Yaskawa INFORM job: CPRINT3D2.JBI

/JOB
//NAME CPRINT3D2
//POS
///NPOS 999,0,0,0,0,0
///TOOL 9
///POSTYPE PULSE
///PULSE
C00000=28439,52447,-122346,62432,-118756,-94394,0
C00001=28774,52172,-123325,61938,-118477,-94718,0
C00002=28786,52165,-123350,61921,-118471,-94727,0
C00003=28820,52146,-123417,61875,-118455,-94751,0
C00004=28874,52134,-123462,61810,-118455,-94770,0
C00005=28928,52121,-123507,61744,-118455,-94790,0
C00006=29088,52031,-123833,61527,-118375,-94904,0
C00007=29175,51999,-123949,61415,-118355,-94948,0
C00008=29421,52045,-123790,61164,-118501,-94935,0
C00009=29495,52038,-123817,61080,-118514,-94952,0
C00010=29569,52031,-123842,60995,-118527,-94969,0
C00011=29587,52039,-123815,60978,-118545,-94964,0
C00012=29506,52029,-123847,61064,-118504,-94962,0
C00013=29829,52073,-123695,60727,-118672,-94961,0
C00014=29932,52093,-123628,60621,-118733,-94956,0
C00015=29996,52105,-123587,60557,-118771,-94953,0
C00016=30178,52149,-123434,60375,-118894,-94933,0
C00017=30236,52166,-123374,60319,-118938,-94924,0
C00018=30330,52195,-123273,60228,-119011,-94908,0
C00019=30378,52209,-123223,60182,-119047,-94901,0
C00020=30588,52286,-122956,59985,-119227,-94854,0
C00021=30620,52321,-122833,59966,-119289,-94824,0
C00022=30635,52338,-122772,59957,-119320,-94809,0
C00023=49239,53005,-120913,62324,-119586,-94086,0
C00024=49295,53006,-120913,62261,-119605,-94093,0
C00025=49352,53006,-120913,62199,-119626,-94101,0
C00026=49357,53007,-120910,62194,-119628,-94101,0
C00027=49400,53018,-120873,62152,-119658,-94096,0
C00028=49596,53097,-120607,61973,-119832,-94048,0
C00029=49625,53101,-120595,61943,-119847,-94048,0
C00030=49712,53113,-120558,61852,-119893,-94050,0
C00031=49739,53123,-120523,61827,-119916,-94044,0
C00032=49769,53136,-120482,61800,-119943,-94037,0
C00033=50226,53391,-119629,61417,-120443,-93863,0
C00034=50247,53407,-119575,61401,-120472,-93851,0
C00035=50264,53421,-119528,61390,-120497,-93840,0
C00036=50275,53464,-119383,61398,-120558,-93801,0
C00037=50279,53479,-119335,61401,-120579,-93788,0
C00038=50414,53586,-118980,61302,-120768,-93708,0
C00039=50453,53638,-118808,61285,-120851,-93666,0
C00040=50279,53728,-118502,61520,-120908,-93555,0
C00041=50270,53764,-118384,61547,-120951,-93521,0
C00042=50261,53800,-118264,61574,-120995,-93487,0
C00043=50239,53805,-118247,61601,-120993,-93478,0
C00044=50284,53772,-118356,61536,-120967,-93516,0
C00045=50093,53900,-117929,61808,-121064,-93368,0
C00046=50021,53939,-117796,61906,-121089,-93320,0
C00047=49977,53963,-117716,61966,-121103,-93291,0
C00048=49831,54030,-117493,62159,-121135,-93207,0
C00049=49779,54050,-117426,62226,-121141,-93181,0
C00050=49693,54082,-117318,62336,-121150,-93137,0
C00051=49650,54098,-117264,62391,-121153,-93116,0
C00052=49433,54167,-117032,62662,-121159,-93019,0
C00053=49353,54169,-117024,62751,-121131,-93005,0
C00054=49313,54170,-117021,62795,-121118,-92998,0
C00055=49104,54236,-116799,63057,-121120,-92904,0
C00056=49064,54233,-116808,63099,-121101,-92901,0
C00057=40018,60732,-97213,75689,-122654,-85947,0
C00058=40054,60785,-97067,75678,-122711,-85911,0
C00059=40032,60817,-96978,75714,-122721,-85882,0
C00060=40014,60842,-96907,75743,-122726,-85859,0
C00061=39996,60867,-96836,75772,-122733,-85836,0
C00062=39979,60893,-96765,75801,-122740,-85813,0
C00063=39961,60918,-96694,75831,-122747,-85790,0
C00064=39951,60933,-96653,75848,-122750,-85776,0
C00065=39894,60999,-96467,75934,-122761,-85715,0
C00066=39865,61033,-96374,75978,-122767,-85684,0
C00067=39823,61077,-96250,76039,-122770,-85642,0
C00068=39761,61137,-96083,76128,-122772,-85585,0
C00069=39725,61172,-95986,76179,-122773,-85552,0
C00070=39700,61192,-95929,76214,-122772,-85532,0
C00071=39675,61212,-95873,76248,-122770,-85512,0
C00072=39649,61232,-95816,76282,-122768,-85492,0
C00073=39624,61253,-95760,76316,-122765,-85472,0
C00074=39598,61273,-95703,76351,-122764,-85452,0
C00075=39580,61287,-95663,76375,-122762,-85438,0
C00076=39514,61268,-95714,76432,-122709,-85443,0
C00077=23111,61906,-93699,72648,-125561,-85469,0
C00078=23063,61952,-93573,72718,-125566,-85425,0
C00079=23022,61942,-93597,72755,-125534,-85425,0
C00080=22989,61935,-93618,72784,-125507,-85426,0
C00081=22956,61927,-93639,72813,-125482,-85426,0
C00082=22923,61919,-93660,72842,-125456,-85426,0
C00083=22890,61912,-93680,72871,-125430,-85426,0
C00084=22871,61907,-93692,72888,-125415,-85427,0
C00085=22781,61878,-93772,72962,-125340,-85434,0
C00086=22736,61863,-93811,73000,-125302,-85438,0
C00087=22678,61841,-93871,73047,-125250,-85445,0
C00088=22634,61823,-93921,73081,-125210,-85452,0
C00089=22547,61786,-94022,73149,-125129,-85466,0
C00090=22530,61777,-94046,73161,-125113,-85470,0
C00091=22501,61761,-94089,73183,-125083,-85477,0
C00092=22472,61745,-94132,73204,-125055,-85484,0
C00093=22442,61729,-94175,73225,-125025,-85492,0
C00094=22413,61713,-94218,73247,-124996,-85499,0
C00095=22377,61694,-94271,73273,-124959,-85508,0
C00096=22378,61632,-94442,73241,-124916,-85557,0
C00097=22087,61535,-94704,73483,-124670,-85584,0
C00098=22099,61276,-95420,73344,-124490,-85788,0
C00099=22144,61093,-95926,73210,-124385,-85939,0
C00100=22157,61056,-96029,73179,-124365,-85970,0
C00101=22183,60982,-96235,73117,-124326,-86033,0
C00102=22199,60937,-96360,73079,-124302,-86071,0
C00103=22261,60808,-96718,72954,-124244,-86182,0
C00104=22286,60767,-96832,72909,-124228,-86219,0
C00105=22328,60702,-97015,72836,-124204,-86278,0
C00106=22437,60560,-97411,72657,-124163,-86407,0
C00107=22476,60515,-97537,72596,-124151,-86449,0
C00108=22493,60521,-97521,72582,-124165,-86447,0
C00109=22439,60543,-97459,72646,-124151,-86421,0
C00110=22493,60521,-97521,72582,-124165,-86447,0
C00111=22546,60499,-97583,72517,-124180,-86474,0
C00112=22546,60446,-97605,72528,-124197,-86456,0
C00113=40139,58675,-102915,74674,-121313,-87587,0
C00114=46748,54147,-116851,65625,-120206,-92552,0
C00115=46543,53843,-117842,65707,-119772,-92808,0
C00116=46527,53787,-118025,65698,-119701,-92859,0
C00117=46489,53721,-118242,65709,-119608,-92917,0
C00118=46439,53445,-119159,65637,-119259,-93176,0
C00119=46497,53175,-120068,65451,-118951,-93447,0
C00120=46664,52922,-120936,65152,-118694,-93722,0
C00121=46813,52797,-121368,64933,-118587,-93867,0
C00122=31513,53470,-118728,59563,-121334,-93793,0
C00123=31001,53645,-118138,60213,-121386,-93553,0
C00124=30898,53667,-118063,60337,-121380,-93517,0
C00125=30785,53702,-117945,60479,-121384,-93467,0
C00126=30275,53799,-117618,61087,-121323,-93299,0
C00127=29739,53845,-117457,61698,-121183,-93173,0
C00128=29195,53838,-117469,62291,-120970,-93095,0
C00129=28904,53806,-117570,62595,-120820,-93080,0
C00130=24595,59466,-100389,69956,-124580,-87578,0
C00131=25008,59807,-99429,69702,-125092,-87378,0
C00132=25274,60150,-98469,69602,-125526,-87155,0
C00133=25393,60407,-97751,69612,-125804,-86976,0
C00134=25484,60702,-96928,69671,-126098,-86762,0
C00135=29736,55171,-113211,83941,-113532,-89553,0
C00136=29662,55374,-112578,84077,-113612,-89348,0
C00137=37622,58900,-102216,77312,-120074,-87045,0
C00138=38136,58667,-102898,76698,-120202,-87311,0
C00139=38618,58542,-103267,76159,-120381,-87482,0
C00140=38958,58510,-103367,75801,-120545,-87556,0
C00141=39335,58507,-103383,75417,-120750,-87612,0
C00142=39839,58581,-103180,74938,-121078,-87622,0
C00143=40057,58649,-102988,74746,-121249,-87596,0
C00144=40323,59480,-100616,74849,-122006,-86947,0
C00145=47960,54217,-116657,64337,-120759,-92670,0
C00146=47759,54094,-117052,64499,-120535,-92753,0
C00147=47571,53923,-117607,64624,-120258,-92884,0
C00148=47451,53740,-118207,64669,-119993,-93039,0
C00149=47440,53697,-118347,64661,-119936,-93078,0
C00150=47411,53644,-118524,64668,-119860,-93124,0
C00151=47383,53460,-119134,64613,-119625,-93296,0
C00152=47428,53280,-119739,64481,-119418,-93476,0
C00153=47544,53111,-120315,64275,-119246,-93657,0
C00154=47729,52958,-120841,64001,-119115,-93834,0
C00155=48077,52776,-121476,63535,-118995,-94063,0
C00156=31284,52867,-120754,59528,-120418,-94315,0
C00157=31125,52990,-120334,59762,-120536,-94176,0
C00158=30851,53126,-119866,60129,-120633,-94006,0
C00159=30540,53231,-119506,60524,-120667,-93860,0
C00160=30461,53248,-119449,60619,-120661,-93833,0
C00161=30368,53276,-119352,60735,-120667,-93793,0
C00162=30024,53340,-119134,61143,-120629,-93682,0
C00163=29662,53370,-119026,61556,-120540,-93598,0
C00164=29294,53365,-119034,61959,-120400,-93547,0
C00165=28932,53327,-119157,62337,-120219,-93530,0
C00166=28454,53226,-119485,62815,-119916,-93555,0
C00167=23569,59757,-99551,71154,-124247,-87172,0
C00168=23875,59858,-99271,70890,-124500,-87143,0
C00169=24154,60011,-98844,70680,-124781,-87070,0
C00170=24390,60208,-98293,70538,-125074,-86955,0
C00171=24575,60444,-97635,70469,-125368,-86801,0
C00172=24652,60608,-97180,70473,-125544,-86687,0
C00173=24715,60805,-96632,70510,-125737,-86544,0
C00174=24738,61093,-95833,70634,-125978,-86325,0
C00175=24696,61382,-95035,70826,-126178,-86094,0
C00176=24554,61763,-93987,71167,-126386,-85776,0
C00177=37748,59756,-99783,77545,-120714,-86351,0
C00178=37941,59542,-100390,77263,-120685,-86553,0
C00179=38191,59363,-100905,76938,-120710,-86736,0
C00180=38484,59228,-101296,76587,-120785,-86889,0
C00181=38809,59142,-101548,76223,-120911,-87006,0
C00182=39022,59121,-101612,76000,-121015,-87054,0
C00183=39270,59119,-101622,75750,-121153,-87090,0
C00184=39611,59170,-101483,75429,-121382,-87097,0
C00185=39931,59273,-101196,75151,-121636,-87059,0
C00186=40250,59441,-100724,74904,-121937,-86968,0
C00187=48252,53381,-119424,63624,-119841,-93498,0
C00188=48319,53287,-119742,63507,-119744,-93599,0
C00189=48423,53202,-120032,63353,-119672,-93696,0
C00190=48560,53129,-120281,63169,-119626,-93786,0
C00191=48724,53072,-120481,62960,-119609,-93865,0
C00192=48911,53031,-120625,62736,-119619,-93932,0
C00193=48970,53025,-120648,62668,-119632,-93947,0
C00194=49055,53010,-120703,62567,-119640,-93974,0
C00195=49583,52969,-120858,61965,-119765,-94091,0
C00196=30650,52240,-122919,59933,-119302,-94827,0
C00197=30671,52456,-122162,60012,-119625,-94618,0
C00198=30635,52559,-121802,60100,-119762,-94512,0
C00199=30555,52657,-121463,60234,-119874,-94406,0
C00200=30442,52741,-121170,60399,-119956,-94309,0
C00201=30291,52816,-120911,60601,-120010,-94215,0
C00202=30117,52874,-120711,60820,-120030,-94134,0
C00203=30060,52885,-120668,60889,-120027,-94115,0
C00204=29985,52907,-120592,60981,-120032,-94083,0
C00205=29793,52942,-120471,61209,-120012,-94021,0
C00206=29591,52959,-120411,61441,-119965,-93976,0
C00207=29384,52956,-120415,61667,-119889,-93948,0
C00208=29182,52935,-120483,61879,-119790,-93939,0
C00209=28992,52896,-120614,62070,-119671,-93949,0
C00210=28820,52840,-120800,62233,-119536,-93978,0
C00211=28673,52771,-121036,62362,-119392,-94025,0
C00212=28639,52747,-121118,62389,-119347,-94043,0
C00213=28578,52715,-121227,62441,-119282,-94066,0
C00214=28300,52499,-121966,62647,-118894,-94240,0
C00215=22491,60387,-97770,72555,-124120,-86493,0
C00216=23005,60287,-98055,71986,-124342,-86658,0
C00217=23190,60283,-98068,71798,-124446,-86691,0
C00218=23373,60311,-97991,71625,-124573,-86699,0
C00219=23550,60370,-97828,71476,-124721,-86683,0
C00220=23711,60460,-97581,71356,-124883,-86640,0
C00221=23849,60576,-97258,71274,-125055,-86572,0
C00222=23959,60716,-96869,71234,-125228,-86481,0
C00223=23997,60795,-96649,71235,-125312,-86426,0
C00224=24033,60905,-96346,71254,-125418,-86347,0
C00225=24049,61076,-95874,71324,-125559,-86217,0
C00226=24026,61246,-95401,71434,-125676,-86080,0
C00227=23966,61411,-94947,71578,-125766,-85942,0
C00228=23918,61488,-94735,71665,-125796,-85875,0
C00229=23843,61582,-94474,71789,-125822,-85788,0
C00230=23703,61701,-94147,71990,-125826,-85672,0
C00231=23297,61933,-93506,72514,-125750,-85423,0
C00232=38223,60782,-96915,77518,-121658,-85582,0
C00233=38238,60338,-98154,77310,-121382,-85943,0
C00234=38280,60189,-98571,77204,-121311,-86070,0
C00235=38359,60050,-98964,77066,-121266,-86195,0
C00236=38471,59925,-99318,76900,-121249,-86312,0
C00237=38616,59820,-99617,76711,-121263,-86419,0
C00238=38786,59741,-99845,76506,-121308,-86508,0
C00239=38976,59689,-99994,76294,-121383,-86578,0
C00240=39078,59679,-100025,76188,-121435,-86601,0
C00241=39213,59678,-100031,76052,-121512,-86621,0
C00242=39412,59709,-99948,75866,-121648,-86625,0
C00243=39600,59770,-99778,75705,-121799,-86602,0
C00244=39770,59860,-99526,75576,-121960,-86554,0
C00245=39843,59919,-99363,75529,-122043,-86517,0
C00246=39927,60004,-99123,75483,-122152,-86460,0
C00247=40019,60149,-98717,75457,-122306,-86356,0
C00248=40157,60547,-97607,75500,-122662,-86056,0
C00249=49381,54129,-116981,62740,-121193,-92971,0
C00250=48940,54060,-117194,63191,-120943,-92965,0
C00251=48744,54006,-117364,63380,-120803,-92984,0
C00252=48573,53936,-117592,63534,-120652,-93024,0
C00253=48434,53851,-117867,63646,-120495,-93082,0
C00254=48330,53756,-118178,63714,-120340,-93155,0
C00255=48266,53654,-118511,63737,-120190,-93240,0
C00256=48259,53624,-118614,63730,-120149,-93269,0
C00257=48237,53581,-118753,63734,-120088,-93305,0
C00258=48225,53480,-119090,63701,-119957,-93400,0
C00259=48238,53430,-119257,63662,-119899,-93449,0
C00260=48103,53311,-119656,63755,-119698,-93544,0
C00261=49484,53946,-117583,62539,-121004,-93155,0
C00262=49610,53938,-117614,62397,-121039,-93182,0
C00263=49860,53921,-117674,62114,-121111,-93237,0
C00264=49874,53920,-117678,62098,-121114,-93240,0
C00265=49888,53919,-117682,62082,-121119,-93243,0
C00266=49902,53918,-117685,62067,-121122,-93246,0
C00267=49916,53917,-117690,62051,-121126,-93249,0
C00268=49930,53916,-117693,62035,-121129,-93252,0
C00269=49942,53915,-117698,62021,-121132,-93255,0
C00270=49954,53913,-117702,62006,-121135,-93259,0
C00271=49967,53912,-117707,61992,-121138,-93262,0
C00272=49979,53911,-117713,61978,-121141,-93265,0
C00273=49991,53909,-117717,61964,-121143,-93268,0
C00274=50002,53908,-117723,61951,-121145,-93271,0
C00275=50014,53906,-117729,61937,-121147,-93274,0
C00276=50026,53905,-117733,61924,-121150,-93278,0
C00277=50037,53903,-117739,61910,-121152,-93281,0
C00278=50049,53902,-117745,61896,-121154,-93284,0
C00279=50061,53900,-117749,61883,-121157,-93288,0
C00280=50123,53870,-117852,61799,-121141,-93325,0
C00281=50159,53851,-117915,61751,-121129,-93348,0
C00282=50186,53835,-117968,61714,-121119,-93367,0
C00283=50213,53819,-118021,61676,-121108,-93386,0
C00284=50240,53803,-118075,61639,-121097,-93405,0
C00285=50267,53787,-118127,61601,-121087,-93424,0
C00286=50285,53775,-118167,61575,-121078,-93437,0
C00287=50303,53763,-118207,61549,-121069,-93451,0
C00288=50319,53753,-118242,61528,-121060,-93464,0
C00289=50334,53742,-118278,61506,-121052,-93476,0
C00290=50349,53731,-118315,61484,-121044,-93488,0
C00291=50364,53721,-118350,61462,-121035,-93500,0
C00292=50379,53710,-118386,61441,-121027,-93512,0
C00293=50394,53699,-118422,61419,-121018,-93524,0
C00294=50407,53690,-118455,61400,-121010,-93536,0
C00295=50418,53681,-118485,61383,-121003,-93545,0
C00296=50429,53672,-118514,61366,-120995,-93555,0
C00297=50441,53663,-118543,61350,-120988,-93566,0
C00298=50450,53655,-118572,61335,-120980,-93575,0
C00299=50460,53646,-118601,61320,-120972,-93584,0
C00300=50470,53637,-118630,61305,-120964,-93594,0
C00301=50479,53629,-118658,61290,-120957,-93603,0
C00302=50489,53620,-118686,61276,-120949,-93613,0
C00303=50498,53613,-118714,61262,-120941,-93621,0
C00304=50506,53605,-118738,61250,-120935,-93629,0
C00305=50513,53598,-118762,61238,-120928,-93637,0
C00306=50521,53591,-118785,61227,-120921,-93645,0
C00307=50527,53584,-118808,61216,-120914,-93652,0
C00308=50534,53578,-118831,61205,-120907,-93659,0
C00309=50544,53567,-118864,61189,-120898,-93670,0
C00310=50538,53559,-118892,61192,-120885,-93677,0
C00311=50531,53550,-118923,61195,-120870,-93684,0
C00312=50524,53541,-118954,61199,-120856,-93692,0
C00313=50517,53531,-118985,61202,-120841,-93699,0
C00314=50509,53522,-119015,61206,-120826,-93707,0
C00315=50500,53511,-119050,61211,-120808,-93715,0
C00316=50491,53501,-119085,61216,-120791,-93724,0
C00317=50481,53491,-119119,61222,-120774,-93732,0
C00318=50472,53480,-119154,61227,-120757,-93740,0
C00319=50463,53470,-119188,61233,-120739,-93748,0
C00320=50453,53459,-119223,61238,-120722,-93757,0
C00321=50444,53449,-119257,61243,-120706,-93765,0
C00322=50433,53438,-119293,61250,-120688,-93773,0
C00323=50422,53428,-119328,61257,-120669,-93782,0
C00324=50411,53417,-119364,61264,-120651,-93790,0
C00325=50396,53404,-119408,61274,-120629,-93800,0
C00326=50378,53388,-119460,61286,-120602,-93812,0
C00327=50360,53372,-119512,61299,-120574,-93823,0
C00328=50342,53357,-119564,61312,-120548,-93836,0
C00329=50323,53341,-119616,61324,-120520,-93847,0
C00330=50301,53324,-119674,61341,-120489,-93860,0
C00331=50271,53302,-119744,61364,-120450,-93876,0
C00332=50234,53278,-119827,61392,-120404,-93894,0
C00333=50198,53253,-119910,61421,-120358,-93912,0
C00334=50189,53251,-119917,61430,-120352,-93912,0
C00335=50178,53249,-119924,61441,-120345,-93912,0
C00336=50167,53246,-119932,61452,-120338,-93913,0
C00337=50156,53244,-119939,61464,-120332,-93913,0
C00338=50144,53242,-119947,61475,-120325,-93914,0
C00339=50133,53239,-119953,61486,-120318,-93914,0
C00340=50120,53237,-119961,61500,-120310,-93914,0
C00341=50106,53235,-119968,61513,-120302,-93914,0
C00342=50093,53232,-119976,61527,-120295,-93915,0
C00343=50080,53230,-119983,61541,-120287,-93915,0
C00344=50067,53228,-119991,61554,-120279,-93915,0
C00345=50053,53225,-119998,61568,-120272,-93915,0
C00346=50040,53223,-120006,61582,-120264,-93916,0
C00347=50026,53221,-120013,61595,-120256,-93916,0
C00348=50013,53218,-120021,61609,-120248,-93916,0
C00349=50000,53216,-120028,61622,-120241,-93916,0
C00350=49986,53214,-120036,61636,-120233,-93916,0
C00351=49973,53211,-120043,61650,-120225,-93916,0
C00352=49887,53199,-120084,61738,-120179,-93916,0
C00353=49729,53176,-120158,61902,-120093,-93914,0
C00354=49571,53153,-120232,62066,-120007,-93912,0
C00355=30261,52244,-122898,60366,-119184,-94767,0
C00356=30138,52138,-123266,60453,-118989,-94854,0
C00357=30073,52083,-123461,60500,-118887,-94901,0
C00358=30066,52078,-123481,60505,-118877,-94906,0
C00359=30059,52072,-123501,60510,-118866,-94910,0
C00360=30051,52066,-123522,60516,-118856,-94915,0
C00361=30044,52061,-123541,60521,-118845,-94919,0
C00362=30037,52055,-123560,60527,-118835,-94924,0
C00363=30030,52050,-123578,60532,-118825,-94928,0
C00364=30023,52045,-123595,60538,-118816,-94932,0
C00365=30015,52040,-123614,60544,-118805,-94936,0
C00366=30008,52036,-123630,60549,-118796,-94940,0
C00367=30001,52031,-123646,60555,-118787,-94943,0
C00368=29993,52027,-123662,60562,-118778,-94947,0
C00369=29986,52022,-123678,60568,-118769,-94951,0
C00370=29979,52017,-123694,60573,-118759,-94954,0
C00371=29971,52013,-123711,60580,-118751,-94958,0
C00372=29964,52008,-123727,60586,-118742,-94961,0
C00373=29960,52006,-123735,60589,-118738,-94964,0
C00374=29919,51997,-123766,60630,-118711,-94967,0
C00375=29852,51983,-123815,60697,-118669,-94972,0
C00376=29807,51975,-123844,60744,-118642,-94974,0
C00377=29765,51968,-123867,60787,-118619,-94975,0
C00378=29724,51961,-123892,60829,-118596,-94976,0
C00379=29683,51954,-123916,60872,-118572,-94978,0
C00380=29647,51948,-123935,60909,-118553,-94979,0
C00381=29617,51944,-123949,60941,-118537,-94979,0
C00382=29588,51940,-123963,60970,-118523,-94979,0
C00383=29561,51937,-123973,60999,-118509,-94979,0
C00384=29534,51934,-123985,61027,-118496,-94978,0
C00385=29507,51931,-123995,61055,-118483,-94977,0
C00386=29481,51928,-124005,61083,-118470,-94977,0
C00387=29454,51924,-124017,61112,-118456,-94977,0
C00388=29427,51921,-124027,61140,-118443,-94976,0
C00389=29405,51919,-124034,61163,-118433,-94976,0
C00390=29383,51917,-124041,61186,-118424,-94975,0
C00391=29361,51915,-124048,61209,-118414,-94974,0
C00392=29340,51913,-124054,61232,-118404,-94973,0
C00393=29320,51912,-124059,61254,-118396,-94972,0
C00394=29299,51910,-124064,61276,-118387,-94971,0
C00395=29279,51909,-124070,61298,-118378,-94969,0
C00396=29258,51907,-124074,61320,-118370,-94968,0
C00397=29237,51906,-124079,61342,-118361,-94967,0
C00398=29220,51905,-124082,61361,-118354,-94965,0
C00399=29203,51904,-124086,61380,-118347,-94964,0
C00400=29185,51903,-124089,61398,-118340,-94963,0
C00401=29169,51902,-124092,61416,-118334,-94962,0
C00402=29153,51901,-124094,61433,-118327,-94960,0
C00403=29137,51900,-124096,61451,-118322,-94959,0
C00404=29121,51900,-124098,61468,-118315,-94958,0
C00405=29099,51908,-124070,61495,-118321,-94947,0
C00406=29084,51914,-124048,61515,-118324,-94938,0
C00407=29068,51919,-124027,61535,-118327,-94930,0
C00408=29053,51926,-124005,61555,-118331,-94922,0
C00409=29037,51932,-123981,61576,-118335,-94913,0
C00410=29020,51939,-123955,61598,-118341,-94903,0
C00411=29003,51946,-123930,61620,-118346,-94894,0
C00412=28986,51954,-123903,61642,-118350,-94884,0
C00413=28969,51961,-123877,61664,-118356,-94875,0
C00414=28952,51968,-123851,61686,-118361,-94865,0
C00415=28935,51975,-123825,61708,-118366,-94855,0
C00416=28918,51982,-123799,61730,-118371,-94846,0
C00417=28901,51990,-123770,61752,-118377,-94835,0
C00418=28884,51998,-123741,61775,-118384,-94824,0
C00419=28867,52007,-123711,61797,-118389,-94814,0
C00420=28843,52019,-123666,61829,-118400,-94798,0
C00421=28819,52032,-123620,61862,-118410,-94782,0
C00422=28795,52044,-123576,61894,-118422,-94766,0
C00423=28772,52057,-123530,61926,-118432,-94749,0
C00424=28747,52071,-123480,61959,-118443,-94732,0
C00425=28721,52086,-123425,61995,-118457,-94713,0
C00426=28685,52109,-123342,62045,-118479,-94684,0
C00427=28650,52133,-123258,62094,-118501,-94656,0
C00428=28632,52146,-123211,62120,-118514,-94640,0
C00429=28632,52152,-123192,62123,-118522,-94635,0
C00430=28632,52157,-123172,62125,-118529,-94629,0
C00431=28632,52162,-123153,62128,-118537,-94624,0
C00432=28631,52168,-123134,62131,-118545,-94618,0
C00433=28631,52173,-123115,62133,-118551,-94612,0
C00434=28631,52179,-123094,62136,-118561,-94606,0
C00435=28632,52185,-123071,62138,-118570,-94600,0
C00436=28633,52192,-123048,62141,-118579,-94593,0
C00437=28633,52198,-123026,62143,-118588,-94587,0
C00438=28634,52205,-123003,62145,-118597,-94581,0
C00439=28634,52211,-122981,62148,-118607,-94574,0
C00440=28635,52217,-122958,62150,-118616,-94568,0
C00441=28635,52224,-122936,62152,-118625,-94561,0
C00442=28636,52230,-122914,62155,-118634,-94555,0
C00443=28636,52237,-122891,62157,-118643,-94549,0
C00444=28637,52243,-122868,62159,-118653,-94542,0
C00445=28637,52249,-122846,62162,-118662,-94536,0
C00446=28638,52256,-122823,62164,-118671,-94530,0
C00447=28652,52331,-122560,62183,-118780,-94456,0
C00448=28666,52406,-122297,62202,-118890,-94383,0
C00449=28673,52444,-122166,62212,-118944,-94346,0
C00450=22620,60686,-96937,72571,-124420,-86279,0
C00451=22593,60700,-96897,72605,-124416,-86262,0
C00452=22539,60729,-96816,72673,-124405,-86231,0
C00453=22508,60746,-96768,72713,-124400,-86213,0
C00454=22499,60752,-96753,72725,-124398,-86207,0
C00455=22489,60758,-96735,72738,-124397,-86200,0
C00456=22478,60765,-96716,72752,-124396,-86193,0
C00457=22468,60772,-96697,72766,-124395,-86186,0
C00458=22458,60779,-96678,72779,-124394,-86179,0
C00459=22448,60785,-96658,72793,-124394,-86171,0
C00460=22437,60792,-96639,72807,-124393,-86164,0
C00461=22427,60799,-96620,72820,-124391,-86157,0
C00462=22417,60806,-96600,72834,-124390,-86150,0
C00463=22406,60813,-96581,72848,-124389,-86143,0
C00464=22397,60819,-96564,72860,-124389,-86137,0
C00465=22389,60825,-96547,72871,-124388,-86131,0
C00466=22381,60831,-96530,72882,-124388,-86125,0
C00467=22373,60837,-96514,72893,-124388,-86119,0
C00468=22366,60844,-96496,72903,-124388,-86112,0
C00469=22358,60850,-96478,72914,-124388,-86106,0
C00470=22350,60856,-96460,72925,-124388,-86100,0
C00471=22342,60863,-96443,72936,-124388,-86094,0
C00472=22335,60869,-96425,72947,-124388,-86087,0
C00473=22327,60875,-96407,72958,-124388,-86081,0
C00474=22319,60882,-96389,72969,-124388,-86074,0
C00475=22311,60888,-96372,72980,-124388,-86069,0
C00476=22304,60895,-96354,72990,-124389,-86062,0
C00477=22296,60901,-96336,73001,-124389,-86056,0
C00478=22288,60907,-96318,73012,-124389,-86049,0
C00479=22281,60914,-96301,73023,-124389,-86043,0
C00480=22274,60920,-96283,73032,-124389,-86037,0
C00481=22267,60926,-96266,73042,-124390,-86031,0
C00482=22260,60932,-96248,73052,-124390,-86025,0
C00483=22253,60939,-96231,73062,-124391,-86019,0
C00484=22247,60945,-96213,73072,-124391,-86013,0
C00485=22240,60951,-96196,73081,-124393,-86007,0
C00486=22234,60957,-96179,73091,-124394,-86001,0
C00487=22228,60963,-96162,73100,-124394,-85996,0
C00488=22222,60970,-96145,73109,-124395,-85990,0
C00489=22216,60976,-96128,73118,-124396,-85984,0
C00490=22210,60982,-96111,73127,-124397,-85978,0
C00491=22207,60985,-96102,73131,-124397,-85975,0
C00492=22203,60998,-96066,73141,-124405,-85964,0
C00493=22196,61024,-95994,73161,-124420,-85943,0
C00494=22191,61048,-95927,73178,-124434,-85923,0
C00495=22186,61070,-95867,73194,-124447,-85905,0
C00496=22181,61092,-95807,73209,-124460,-85888,0
C00497=22179,61111,-95754,73221,-124472,-85872,0
C00498=22176,61130,-95701,73233,-124485,-85857,0
C00499=22173,61149,-95649,73245,-124496,-85841,0
C00500=22170,61168,-95596,73258,-124509,-85826,0
C00501=22167,61187,-95543,73270,-124520,-85810,0
C00502=22165,61203,-95499,73279,-124532,-85798,0
C00503=22164,61219,-95453,73289,-124542,-85784,0
C00504=22162,61236,-95408,73298,-124554,-85772,0
C00505=22161,61252,-95363,73308,-124564,-85758,0
C00506=22160,61266,-95324,73315,-124574,-85747,0
C00507=22160,61280,-95285,73323,-124583,-85736,0
C00508=22159,61295,-95246,73330,-124594,-85725,0
C00509=22159,61309,-95207,73337,-124604,-85714,0
C00510=22158,61323,-95167,73345,-124613,-85702,0
C00511=22158,61337,-95128,73353,-124624,-85691,0
C00512=22157,61352,-95089,73360,-124634,-85680,0
C00513=22157,61364,-95053,73367,-124643,-85670,0
C00514=22157,61377,-95018,73373,-124652,-85660,0
C00515=22157,61390,-94982,73379,-124662,-85650,0
C00516=22162,61395,-94970,73376,-124667,-85647,0
C00517=22173,61404,-94946,73370,-124680,-85642,0
C00518=22183,61412,-94922,73364,-124693,-85637,0
C00519=22195,61422,-94896,73357,-124706,-85632,0
C00520=22207,61431,-94870,73350,-124721,-85626,0
C00521=22219,61441,-94844,73342,-124735,-85621,0
C00522=22231,61450,-94818,73335,-124749,-85615,0
C00523=22243,61460,-94792,73328,-124763,-85610,0
C00524=22255,61469,-94766,73320,-124778,-85604,0
C00525=22267,61479,-94740,73313,-124791,-85599,0
C00526=22280,61489,-94713,73305,-124806,-85593,0
C00527=22294,61499,-94685,73296,-124822,-85588,0
C00528=22309,61509,-94656,73286,-124840,-85582,0
C00529=22323,61520,-94628,73277,-124856,-85577,0
C00530=22338,61530,-94599,73267,-124872,-85571,0
C00531=22354,61541,-94571,73257,-124889,-85566,0
C00532=22367,61549,-94547,73248,-124903,-85561,0
C00533=22376,61557,-94527,73243,-124914,-85557,0
C00534=22391,61567,-94499,73233,-124930,-85551,0
C00535=22407,61577,-94470,73223,-124948,-85546,0
C00536=22422,61588,-94442,73213,-124965,-85540,0
C00537=22440,61600,-94410,73201,-124983,-85534,0
C00538=22460,61612,-94375,73186,-125005,-85528,0
C00539=22481,61625,-94340,73172,-125027,-85521,0
C00540=22501,61638,-94306,73158,-125049,-85514,0
C00541=22522,61651,-94271,73144,-125071,-85508,0
C00542=22547,61665,-94233,73126,-125096,-85502,0
C00543=22572,61679,-94194,73108,-125121,-85495,0
C00544=22604,61695,-94150,73084,-125153,-85488,0
C00545=22621,61703,-94128,73072,-125168,-85484,0
C00546=22625,61703,-94128,73067,-125172,-85485,0
C00547=22634,61703,-94127,73059,-125178,-85486,0
C00548=22643,61704,-94127,73050,-125183,-85488,0
C00549=22653,61704,-94126,73041,-125189,-85489,0
C00550=22662,61704,-94126,73032,-125195,-85491,0
C00551=22671,61704,-94125,73023,-125200,-85492,0
C00552=22680,61704,-94125,73014,-125206,-85493,0
C00553=22689,61705,-94124,73005,-125212,-85495,0
C00554=22699,61704,-94125,72994,-125218,-85496,0
C00555=22710,61704,-94126,72984,-125223,-85498,0
C00556=22720,61704,-94126,72974,-125230,-85501,0
C00557=22730,61704,-94127,72963,-125236,-85502,0
C00558=22740,61704,-94128,72953,-125242,-85504,0
C00559=22752,61703,-94130,72942,-125249,-85506,0
C00560=22763,61702,-94132,72930,-125256,-85509,0
C00561=22774,61702,-94134,72918,-125261,-85512,0
C00562=22786,61701,-94136,72907,-125268,-85514,0
C00563=22797,61700,-94138,72895,-125274,-85517,0
C00564=22808,61699,-94141,72883,-125281,-85519,0
C00565=22820,61699,-94143,72872,-125287,-85521,0
C00566=22831,61698,-94145,72860,-125294,-85524,0
C00567=22842,61697,-94147,72848,-125299,-85527,0
C00568=22854,61696,-94149,72837,-125306,-85529,0
C00569=22865,61696,-94151,72825,-125313,-85531,0
C00570=22937,61688,-94172,72749,-125351,-85550,0
C00571=23071,61674,-94213,72609,-125422,-85584,0
C00572=23204,61660,-94252,72469,-125494,-85617,0
C00573=38596,60759,-96984,77141,-121870,-85654,0
C00574=38614,60811,-96839,77146,-121914,-85614,0
C00575=38632,60864,-96695,77151,-121959,-85575,0
C00576=38636,60873,-96669,77152,-121968,-85568,0
C00577=38640,60882,-96643,77152,-121976,-85561,0
C00578=38645,60893,-96614,77152,-121985,-85554,0
C00579=38650,60903,-96585,77151,-121996,-85546,0
C00580=38655,60914,-96556,77151,-122005,-85538,0
C00581=38660,60924,-96527,77151,-122015,-85531,0
C00582=38665,60934,-96499,77151,-122024,-85523,0
C00583=38670,60945,-96470,77151,-122035,-85516,0
C00584=38675,60955,-96441,77150,-122044,-85508,0
C00585=38680,60966,-96412,77150,-122053,-85500,0
C00586=38684,60976,-96383,77150,-122063,-85492,0
C00587=38689,60985,-96360,77149,-122071,-85487,0
C00588=38693,60993,-96337,77148,-122079,-85481,0
C00589=38698,61001,-96314,77148,-122087,-85474,0
C00590=38703,61009,-96291,77147,-122095,-85469,0
C00591=38708,61018,-96268,77145,-122104,-85463,0
C00592=38713,61026,-96246,77144,-122113,-85457,0
C00593=38718,61034,-96223,77143,-122121,-85451,0
C00594=38723,61042,-96200,77142,-122129,-85445,0
C00595=38728,61051,-96177,77140,-122137,-85440,0
C00596=38733,61059,-96155,77139,-122146,-85433,0
C00597=38738,61067,-96132,77138,-122154,-85427,0
C00598=38743,61076,-96109,77137,-122162,-85422,0
C00599=38748,61084,-96086,77136,-122170,-85416,0
C00600=38753,61092,-96063,77134,-122179,-85410,0
C00601=38758,61100,-96041,77133,-122187,-85404,0
C00602=38763,61108,-96020,77131,-122195,-85399,0
C00603=38768,61115,-95999,77130,-122204,-85394,0
C00604=38773,61123,-95979,77128,-122212,-85389,0
C00605=38778,61130,-95958,77126,-122218,-85383,0
C00606=38783,61138,-95937,77125,-122226,-85378,0
C00607=38788,61145,-95916,77123,-122235,-85373,0
C00608=38793,61152,-95898,77121,-122243,-85368,0
C00609=38798,61159,-95879,77119,-122249,-85363,0
C00610=38804,61166,-95860,77117,-122258,-85358,0
C00611=38809,61173,-95841,77115,-122264,-85354,0
C00612=38814,61179,-95822,77113,-122272,-85349,0
C00613=38819,61186,-95803,77111,-122279,-85344,0
C00614=38846,61200,-95767,77091,-122305,-85337,0
C00615=38873,61213,-95730,77071,-122330,-85331,0
C00616=38895,61224,-95702,77053,-122351,-85326,0
C00617=38918,61234,-95675,77035,-122371,-85321,0
C00618=38939,61243,-95650,77019,-122390,-85317,0
C00619=38959,61251,-95628,77003,-122407,-85314,0
C00620=38979,61259,-95607,76986,-122424,-85311,0
C00621=38999,61267,-95585,76970,-122443,-85307,0
C00622=39019,61275,-95563,76954,-122460,-85304,0
C00623=39038,61282,-95544,76939,-122476,-85301,0
C00624=39055,61288,-95528,76925,-122490,-85299,0
C00625=39073,61294,-95511,76911,-122505,-85296,0
C00626=39090,61300,-95495,76896,-122520,-85294,0
C00627=39106,61305,-95480,76883,-122532,-85292,0
C00628=39122,61310,-95468,76870,-122545,-85291,0
C00629=39137,61315,-95456,76857,-122557,-85290,0
C00630=39152,61319,-95443,76844,-122570,-85288,0
C00631=39167,61324,-95430,76831,-122582,-85287,0
C00632=39183,61328,-95418,76819,-122594,-85285,0
C00633=39198,61333,-95405,76806,-122607,-85284,0
C00634=39213,61337,-95394,76793,-122618,-85283,0
C00635=39226,61341,-95383,76781,-122630,-85282,0
C00636=39247,61347,-95368,76763,-122646,-85280,0
C00637=39260,61341,-95386,76748,-122649,-85288,0
C00638=39273,61334,-95403,76733,-122653,-85294,0
C00639=39285,61328,-95422,76718,-122656,-85302,0
C00640=39299,61321,-95442,76701,-122661,-85309,0
C00641=39312,61313,-95463,76684,-122664,-85317,0
C00642=39326,61306,-95483,76667,-122668,-85325,0
C00643=39340,61298,-95504,76651,-122671,-85333,0
C00644=39354,61291,-95525,76634,-122675,-85341,0
C00645=39367,61284,-95545,76617,-122678,-85349,0
C00646=39381,61276,-95566,76600,-122682,-85357,0
C00647=39396,61267,-95591,76581,-122685,-85366,0
C00648=39412,61258,-95617,76562,-122688,-85376,0
C00649=39427,61249,-95642,76543,-122692,-85385,0
C00650=39442,61240,-95668,76524,-122695,-85395,0
C00651=39458,61230,-95697,76504,-122699,-85405,0
C00652=39473,61219,-95726,76484,-122701,-85416,0
C00653=39484,61213,-95742,76471,-122703,-85422,0
C00654=39497,61205,-95764,76454,-122707,-85430,0
C00655=39512,61196,-95792,76434,-122710,-85441,0
C00656=39528,61186,-95819,76415,-122713,-85451,0
C00657=39544,61176,-95846,76395,-122716,-85461,0
C00658=39563,61162,-95884,76369,-122719,-85474,0
C00659=39583,61149,-95922,76344,-122722,-85488,0
C00660=39602,61135,-95960,76319,-122725,-85502,0
C00661=39622,61122,-95998,76293,-122728,-85516,0
C00662=39643,61106,-96041,76265,-122731,-85531,0
C00663=39665,61089,-96088,76236,-122732,-85548,0
C00664=39689,61070,-96144,76203,-122734,-85568,0
C00665=39716,61047,-96208,76166,-122736,-85590,0
C00666=39719,61039,-96230,76159,-122732,-85597,0
C00667=39722,61031,-96253,76152,-122729,-85604,0
C00668=39725,61022,-96275,76146,-122725,-85611,0
C00669=39728,61014,-96298,76139,-122722,-85618,0
C00670=39731,61006,-96321,76132,-122717,-85625,0
C00671=39734,60998,-96343,76126,-122714,-85632,0
C00672=39737,60990,-96366,76119,-122710,-85639,0
C00673=39740,60981,-96390,76112,-122707,-85646,0
C00674=39743,60973,-96414,76106,-122702,-85653,0
C00675=39745,60964,-96438,76099,-122698,-85660,0
C00676=39748,60955,-96462,76093,-122694,-85668,0
C00677=39751,60947,-96486,76086,-122690,-85675,0
C00678=39753,60938,-96510,76080,-122685,-85682,0
C00679=39755,60929,-96536,76073,-122680,-85690,0
C00680=39758,60920,-96561,76067,-122676,-85698,0
C00681=39760,60910,-96587,76061,-122671,-85705,0
C00682=39762,60901,-96612,76054,-122667,-85713,0
C00683=39764,60892,-96638,76048,-122662,-85720,0
C00684=39767,60883,-96664,76041,-122656,-85729,0
C00685=39769,60873,-96690,76034,-122652,-85736,0
C00686=39772,60864,-96715,76028,-122647,-85744,0
C00687=39774,60855,-96741,76021,-122642,-85752,0
C00688=39776,60846,-96767,76015,-122638,-85759,0
C00689=39779,60836,-96793,76008,-122633,-85767,0
C00690=39798,60741,-97060,75946,-122580,-85847,0
C00691=39817,60645,-97326,75883,-122526,-85926,0
C00692=39836,60550,-97593,75821,-122474,-86005,0
C00693=45682,53138,-120172,66324,-118610,-93372,0
C00694=45674,52645,-121863,66111,-117998,-93869,0
C00695=44634,52188,-123439,67047,-117062,-94214,0
C00696=44758,54796,-114715,68077,-120115,-91658,0
C00697=43851,55342,-112973,69298,-120283,-91026,0
C00698=43558,51754,-124971,68039,-116147,-94558,0
C00699=35828,55385,-112658,55729,-125484,-92925,0
C00700=42972,55913,-111183,70491,-120437,-90384,0
C00701=42122,56509,-109345,71656,-120579,-89732,0
C00702=34741,54943,-114022,56714,-124489,-93077,0
C00703=33627,54523,-115336,57740,-123516,-93225,0
C00704=41299,57132,-107459,72794,-120707,-89069,0
C00705=40502,57781,-105522,73906,-120825,-88394,0
C00706=32484,54123,-116600,58808,-122563,-93371,0
C00707=31422,53778,-117706,59814,-121717,-93500,0
C00708=31343,53805,-117615,59913,-121724,-93463,0
C00709=39703,58271,-104075,74939,-120775,-87864,0
C00710=39453,58235,-104175,75179,-120613,-87859,0
C00711=38947,58238,-104155,75695,-120342,-87786,0
C00712=38835,58249,-104123,75814,-120289,-87761,0
C00713=30443,54000,-116963,60999,-121645,-93144,0
C00714=30386,54011,-116927,61067,-121638,-93125,0
C00715=29676,54073,-116711,61877,-121449,-92957,0
C00716=29483,54070,-116716,62087,-121372,-92929,0
C00717=37998,58405,-103651,76727,-119943,-87514,0
C00718=37843,58446,-103530,76900,-119886,-87458,0
C00719=37729,58497,-103381,77037,-119858,-87400,0
C00720=37077,58138,-104410,77547,-119252,-87621,0
C00721=28767,54578,-115071,63115,-121708,-92361,0
C00722=28148,55245,-112953,64110,-122225,-91675,0
C00723=36080,57620,-105905,78347,-118358,-87945,0
C00724=35060,57126,-107348,79190,-117482,-88260,0
C00725=27554,55941,-110793,65090,-122730,-90978,0
C00726=26983,56666,-108586,66059,-123222,-90270,0
C00727=34014,56655,-108740,80077,-116621,-88568,0
C00728=32944,56205,-110079,81006,-115777,-88868,0
C00729=26433,57420,-106332,67016,-123702,-89550,0
C00730=25904,58204,-104028,67965,-124172,-88817,0
C00731=31848,55777,-111368,81977,-114950,-89160,0
C00732=30753,55380,-112578,82967,-114158,-89439,0
C00733=30770,55088,-113489,82859,-113987,-89725,0
C00734=30680,54776,-114473,82855,-113749,-90025,0
C00735=26127,60200,-98338,68749,-126045,-87270,0
C00736=25784,59746,-99612,68869,-125469,-87564,0
C00737=25695,59670,-99827,68922,-125356,-87608,0
C00738=25394,59020,-101671,68905,-124633,-88072,0
C00739=25394,58965,-101693,68916,-124652,-88054,0
C00740=46773,54075,-116914,65603,-120227,-92547,0
C00741=46546,53811,-117769,65727,-119832,-92761,0
C00742=46418,53530,-118693,65737,-119451,-93011,0
C00743=46401,53246,-119643,65626,-119103,-93284,0
C00744=46500,52969,-120579,65391,-118800,-93570,0
C00745=46732,52695,-121525,65013,-118534,-93876,0
C00746=31484,53400,-118780,59600,-121340,-93778,0
C00747=31055,53575,-118189,60159,-121423,-93551,0
C00748=30561,53710,-117739,60769,-121420,-93351,0
C00749=30022,53794,-117452,61402,-121329,-93189,0
C00750=29460,53824,-117345,62033,-121155,-93074,0
C00751=28851,53796,-117424,62687,-120890,-93006,0
C00752=24602,59401,-100443,69954,-124593,-87570,0
C00753=24956,59713,-99564,69746,-125049,-87384,0
C00754=25208,60061,-98589,69664,-125477,-87154,0
C00755=25366,60447,-97511,69699,-125884,-86880,0
C00756=25428,60854,-96382,69846,-126249,-86576,0
C00757=29578,55287,-112687,84160,-113567,-89347,0
C00758=37609,58838,-102260,77331,-120076,-87031,0
C00759=38075,58642,-102833,76781,-120204,-87259,0
C00760=38560,58530,-103166,76245,-120395,-87419,0
C00761=39066,58496,-103274,75719,-120650,-87519,0
C00762=39565,58541,-103155,75232,-120957,-87552,0
C00763=40083,58671,-102789,74763,-121337,-87517,0
C00764=46701,54111,-116794,65697,-120241,-92503,0
C00765=47982,54146,-116714,64319,-120780,-92663,0
C00766=47672,53932,-117402,64556,-120406,-92814,0
C00767=47610,53867,-117614,64593,-120305,-92865,0
C00768=47581,53845,-117685,64615,-120267,-92882,0
C00769=47432,53669,-118262,64695,-119998,-93026,0
C00770=47352,53481,-118881,64695,-119741,-93192,0
C00771=47346,53290,-119518,64613,-119504,-93375,0
C00772=47419,53104,-120147,64447,-119297,-93566,0
C00773=47570,52930,-120742,64202,-119130,-93757,0
C00774=47794,52776,-121276,63884,-119008,-93941,0
C00775=48011,52680,-121614,63602,-118955,-94067,0
C00776=31261,52798,-120800,59559,-120429,-94299,0
C00777=30954,52999,-120113,59995,-120605,-94064,0
C00778=30850,53045,-119956,60132,-120633,-94005,0
C00779=30816,53065,-119888,60178,-120649,-93982,0
C00780=30527,53182,-119489,60553,-120706,-93829,0
C00781=30193,53270,-119186,60963,-120707,-93695,0
C00782=29827,53326,-118993,61393,-120650,-93588,0
C00783=29443,53346,-118920,61825,-120536,-93511,0
C00784=29054,53329,-118971,62244,-120372,-93469,0
C00785=28674,53274,-119148,62634,-120163,-93464,0
C00786=28410,53206,-119367,62893,-119979,-93489,0
C00787=23596,59651,-99721,71111,-124239,-87200,0
C00788=23815,59731,-99500,70926,-124425,-87174,0
C00789=24092,59893,-99047,70723,-124712,-87092,0
C00790=24322,60097,-98477,70590,-125006,-86970,0
C00791=24495,60335,-97812,70533,-125296,-86814,0
C00792=24606,60598,-97081,70553,-125569,-86627,0
C00793=24652,60874,-96317,70647,-125814,-86421,0
C00794=24634,61151,-95550,70808,-126021,-86204,0
C00795=24554,61425,-94794,71031,-126184,-85978,0
C00796=24424,61658,-94153,71282,-126285,-85776,0
C00797=37692,59667,-99901,77596,-120674,-86353,0
C00798=37839,59517,-100329,77387,-120660,-86497,0
C00799=38099,59341,-100833,77053,-120694,-86678,0
C00800=38398,59213,-101205,76699,-120779,-86826,0
C00801=38724,59135,-101432,76339,-120911,-86936,0
C00802=39062,59112,-101505,75989,-121085,-87003,0
C00803=39396,59143,-101425,75667,-121296,-87025,0
C00804=39711,59224,-101199,75385,-121531,-87005,0
C00805=39998,59353,-100837,75154,-121785,-86940,0
C00806=40229,59515,-100382,74993,-122033,-86842,0
C00807=47909,54182,-116597,64415,-120793,-92619,0
C00808=48187,53337,-119385,63713,-119866,-93452,0
C00809=48232,53232,-119741,63615,-119748,-93560,0
C00810=48320,53132,-120079,63472,-119652,-93668,0
C00811=48450,53043,-120386,63287,-119582,-93774,0
C00812=48618,52967,-120646,63067,-119542,-93871,0
C00813=48819,52909,-120849,62819,-119535,-93957,0
C00814=49045,52872,-120984,62553,-119563,-94026,0
C00815=49468,52844,-121090,62073,-119670,-94115,0
C00816=30478,52131,-123098,60113,-119210,-94827,0
C00817=30569,52373,-122254,60124,-119591,-94603,0
C00818=30563,52468,-121923,60176,-119726,-94510,0
C00819=30516,52561,-121599,60271,-119843,-94413,0
C00820=30430,52649,-121295,60408,-119939,-94316,0
C00821=30311,52727,-121024,60576,-120007,-94224,0
C00822=30223,52766,-120891,60691,-120032,-94174,0
C00823=30205,52777,-120853,60716,-120041,-94161,0
C00824=30044,52841,-120631,60925,-120074,-94076,0
C00825=29856,52890,-120461,61155,-120075,-94001,0
C00826=29647,52921,-120352,61399,-120045,-93941,0
C00827=29427,52932,-120311,61647,-119982,-93899,0
C00828=29202,52922,-120340,61890,-119890,-93875,0
C00829=28981,52891,-120442,62118,-119771,-93873,0
C00830=28773,52839,-120613,62322,-119628,-93892,0
C00831=28587,52768,-120851,62495,-119469,-93934,0
C00832=28430,52682,-121146,62626,-119298,-93997,0
C00833=28219,52507,-121744,62778,-118989,-94139,0
C00834=22561,60189,-98196,72425,-124069,-86601,0
C00835=23048,60150,-98311,71913,-124320,-86713,0
C00836=23247,60168,-98264,71720,-124448,-86732,0
C00837=23408,60210,-98148,71578,-124573,-86725,0
C00838=23468,60232,-98087,71527,-124626,-86718,0
C00839=23631,60329,-97819,71410,-124795,-86670,0
C00840=23766,60449,-97485,71333,-124966,-86598,0
C00841=23867,60588,-97099,71300,-125134,-86507,0
C00842=23933,60741,-96677,71310,-125290,-86399,0
C00843=23961,60899,-96238,71361,-125429,-86280,0
C00844=23953,61057,-95801,71449,-125545,-86156,0
C00845=23910,61210,-95377,71571,-125637,-86030,0
C00846=23837,61347,-95000,71713,-125697,-85911,0
C00847=23733,61472,-94655,71882,-125728,-85796,0
C00848=23658,61531,-94492,71986,-125728,-85738,0
C00849=23644,61546,-94449,72009,-125730,-85723,0
C00850=23515,61639,-94192,72185,-125721,-85629,0
C00851=23137,61819,-93697,72653,-125622,-85426,0
C00852=38075,60632,-97204,77630,-121522,-85621,0
C00853=38152,60228,-98332,77380,-121309,-85958,0
C00854=38223,60074,-98767,77244,-121251,-86094,0
C00855=38312,59956,-99098,77105,-121227,-86202,0
C00856=38353,59914,-99217,77046,-121223,-86242,0
C00857=38506,59810,-99514,76849,-121243,-86349,0
C00858=38680,59734,-99732,76643,-121293,-86436,0
C00859=38867,59689,-99864,76436,-121372,-86500,0
C00860=39060,59675,-99906,76238,-121474,-86539,0
C00861=39249,59693,-99860,76057,-121596,-86552,0
C00862=39427,59740,-99731,75899,-121731,-86540,0
C00863=39587,59813,-99527,75771,-121875,-86503,0
C00864=39724,59910,-99257,75678,-122021,-86445,0
C00865=39833,60025,-98934,75621,-122164,-86367,0
C00866=39877,60101,-98722,75611,-122243,-86312,0
C00867=39891,60117,-98678,75605,-122261,-86301,0
C00868=39957,60248,-98313,75598,-122391,-86206,0
C00869=40045,60609,-97306,75675,-122690,-85929,0
C00870=49522,54005,-117217,62565,-121192,-93032,0
C00871=49009,53959,-117353,63105,-120944,-92995,0
C00872=48821,53922,-117469,63295,-120828,-92999,0
C00873=48648,53867,-117644,63457,-120696,-93023,0
C00874=48499,53796,-117871,63588,-120553,-93066,0
C00875=48377,53713,-118142,63681,-120405,-93125,0
C00876=48326,53658,-118321,63711,-120319,-93169,0
C00877=48310,53646,-118361,63724,-120297,-93177,0
C00878=48229,53549,-118681,63766,-120147,-93258,0
C00879=48187,53444,-119027,63763,-120002,-93350,0
C00880=48187,53388,-119217,63736,-119930,-93404,0
C00881=48008,53272,-119598,63879,-119720,-93488,0
C00882=49646,53783,-117948,62322,-120960,-93255,0
C00883=49711,53778,-117965,62248,-120977,-93270,0
C00884=49784,53772,-117986,62165,-120997,-93287,0
C00885=49798,53770,-117992,62149,-121000,-93291,0
C00886=49812,53769,-117998,62133,-121003,-93294,0
C00887=49825,53767,-118004,62117,-121005,-93298,0
C00888=49839,53765,-118010,62101,-121008,-93302,0
C00889=49853,53763,-118017,62084,-121011,-93306,0
C00890=49869,53761,-118024,62066,-121014,-93310,0
C00891=49884,53759,-118031,62048,-121018,-93314,0
C00892=49900,53757,-118038,62030,-121021,-93318,0
C00893=49916,53755,-118045,62012,-121023,-93323,0
C00894=49931,53754,-118052,61994,-121027,-93327,0
C00895=49947,53752,-118058,61976,-121030,-93331,0
C00896=49960,53750,-118065,61961,-121033,-93335,0
C00897=49973,53748,-118071,61946,-121035,-93339,0
C00898=49985,53746,-118078,61931,-121036,-93342,0
C00899=49998,53744,-118086,61916,-121038,-93346,0
C00900=50010,53741,-118093,61901,-121039,-93350,0
C00901=50022,53739,-118101,61887,-121042,-93354,0
C00902=50035,53737,-118109,61872,-121043,-93359,0
C00903=50047,53735,-118117,61858,-121045,-93363,0
C00904=50059,53732,-118124,61843,-121046,-93366,0
C00905=50071,53730,-118132,61828,-121047,-93370,0
C00906=50084,53728,-118140,61814,-121050,-93374,0
C00907=50096,53726,-118147,61799,-121051,-93378,0
C00908=50108,53723,-118155,61785,-121052,-93382,0
C00909=50121,53721,-118163,61770,-121054,-93386,0
C00910=50133,53719,-118171,61755,-121055,-93390,0
C00911=50145,53717,-118178,61741,-121058,-93394,0
C00912=50156,53715,-118186,61728,-121058,-93398,0
C00913=50166,53712,-118193,61715,-121059,-93401,0
C00914=50177,53710,-118201,61703,-121060,-93405,0
C00915=50187,53708,-118209,61690,-121061,-93409,0
C00916=50198,53706,-118216,61677,-121062,-93412,0
C00917=50208,53704,-118224,61665,-121064,-93417,0
C00918=50218,53701,-118232,61652,-121064,-93420,0
C00919=50228,53699,-118240,61640,-121065,-93424,0
C00920=50238,53697,-118248,61628,-121065,-93428,0
C00921=50243,53695,-118252,61622,-121065,-93429,0
C00922=50254,53689,-118275,61607,-121060,-93437,0
C00923=50276,53675,-118319,61577,-121051,-93453,0
C00924=50297,53661,-118365,61546,-121041,-93469,0
C00925=50319,53648,-118410,61516,-121031,-93485,0
C00926=50334,53637,-118446,61494,-121022,-93497,0
C00927=50349,53627,-118481,61472,-121014,-93509,0
C00928=50365,53616,-118516,61450,-121006,-93521,0
C00929=50378,53606,-118550,61431,-120998,-93533,0
C00930=50391,53596,-118584,61412,-120989,-93544,0
C00931=50404,53586,-118617,61392,-120981,-93555,0
C00932=50417,53576,-118650,61373,-120973,-93566,0
C00933=50430,53566,-118685,61354,-120964,-93577,0
C00934=50443,53556,-118718,61335,-120956,-93589,0
C00935=50455,53547,-118748,61318,-120947,-93599,0
C00936=50464,53539,-118776,61303,-120941,-93608,0
C00937=50474,53531,-118803,61288,-120933,-93617,0
C00938=50484,53523,-118831,61274,-120926,-93627,0
C00939=50494,53514,-118859,61259,-120918,-93635,0
C00940=50505,53504,-118893,61242,-120908,-93646,0
C00941=50500,53496,-118920,61244,-120896,-93653,0
C00942=50495,53488,-118947,61245,-120883,-93660,0
C00943=50489,53480,-118974,61247,-120870,-93667,0
C00944=50484,53471,-119001,61249,-120858,-93674,0
C00945=50479,53463,-119028,61250,-120846,-93681,0
C00946=50474,53455,-119055,61252,-120834,-93687,0
C00947=50469,53447,-119082,61254,-120821,-93694,0
C00948=50464,53439,-119109,61256,-120808,-93701,0
C00949=50459,53431,-119136,61258,-120796,-93707,0
C00950=50452,53422,-119166,61261,-120781,-93715,0
C00951=50445,53413,-119196,61264,-120767,-93722,0
C00952=50439,53404,-119225,61267,-120753,-93729,0
C00953=50432,53395,-119255,61270,-120738,-93736,0
C00954=50424,53386,-119286,61274,-120723,-93744,0
C00955=50416,53375,-119320,61279,-120707,-93753,0
C00956=50407,53365,-119354,61283,-120690,-93760,0
C00957=50398,53355,-119387,61288,-120674,-93768,0
C00958=50389,53345,-119420,61293,-120658,-93776,0
C00959=50380,53335,-119455,61298,-120641,-93784,0
C00960=50372,53325,-119488,61303,-120625,-93793,0
C00961=50363,53315,-119521,61308,-120608,-93801,0
C00962=50353,53305,-119555,61314,-120591,-93809,0
C00963=50343,53295,-119588,61320,-120575,-93816,0
C00964=50333,53285,-119621,61326,-120558,-93824,0
C00965=50317,53271,-119668,61337,-120533,-93835,0
C00966=50301,53256,-119717,61348,-120508,-93846,0
C00967=50284,53242,-119764,61360,-120483,-93857,0
C00968=50268,53228,-119811,61371,-120459,-93868,0
C00969=50252,53213,-119859,61382,-120434,-93879,0
C00970=50232,53198,-119912,61396,-120406,-93891,0
C00971=50206,53178,-119975,61416,-120372,-93905,0
C00972=50174,53156,-120051,61441,-120330,-93921,0
C00973=50142,53134,-120126,61465,-120289,-93938,0
C00974=50112,53113,-120192,61489,-120252,-93952,0
C00975=50100,53111,-120201,61501,-120244,-93953,0
C00976=50088,53108,-120209,61513,-120237,-93953,0
C00977=50077,53106,-120217,61524,-120229,-93954,0
C00978=50065,53104,-120224,61536,-120222,-93954,0
C00979=50053,53102,-120232,61549,-120215,-93954,0
C00980=50039,53099,-120238,61562,-120207,-93955,0
C00981=50025,53097,-120246,61577,-120199,-93955,0
C00982=50011,53095,-120253,61592,-120191,-93955,0
C00983=49996,53092,-120261,61607,-120183,-93955,0
C00984=49981,53090,-120269,61622,-120175,-93955,0
C00985=49966,53087,-120276,61637,-120167,-93955,0
C00986=49951,53085,-120284,61653,-120158,-93955,0
C00987=49936,53083,-120292,61668,-120150,-93955,0
C00988=49922,53080,-120299,61683,-120142,-93955,0
C00989=49907,53078,-120307,61698,-120134,-93955,0
C00990=49892,53076,-120314,61714,-120126,-93955,0
C00991=49877,53073,-120322,61729,-120117,-93955,0
C00992=49691,53048,-120402,61922,-120020,-93951,0
C00993=49505,53024,-120479,62116,-119924,-93947,0
C00994=30005,52138,-123063,60640,-119069,-94753,0
C00995=29937,52084,-123254,60689,-118967,-94798,0
C00996=29928,52077,-123278,60696,-118955,-94803,0
C00997=29918,52071,-123300,60704,-118942,-94808,0
C00998=29909,52065,-123322,60712,-118930,-94813,0
//INST
///DATE 2025/02/20 16:20
///COMM Generated using RoboDK
///ATTR SC,RW
///GROUP1 RB1
NOP
MOVL C00000 V=30.0 PL=1
CALL JOB:EXTRUDE
CALL JOB:EXTRUDE
MOVL C00001 V=130.0 PL=1
CALL JOB:EXTRUDE
CALL JOB:EXTRUDE
MOVL C00002 V=30.0 PL=1
CALL JOB:EXTRUDE
MOVL C00003 V=30.0 PL=1
CALL JOB:EXTRUDE
MOVL C00004 V=30.0 PL=1
CALL JOB:EXTRUDE
MOVL C00005 V=30.0 PL=1
MOVL C00006 V=130.0 PL=1
CALL JOB:EXTRUDE
MOVL C00007 V=30.0 PL=1
MOVL C00008 V=130.0 PL=1
CALL JOB:EXTRUDE
MOVL C00009 V=30.0 PL=1
CALL JOB:EXTRUDE
MOVL C00010 V=30.0 PL=1
MOVL C00011 V=130.0 PL=1
CALL JOB:EXTRUDE
MOVL C00012 V=30.0 PL=1
CALL JOB:EXTRUDE
CALL JOB:EXTRUDE
MOVL C00013 V=130.0 PL=1
CALL JOB:EXTRUDE
CALL JOB:EXTRUDE
MOVL C00014 V=30.0 PL=1
CALL JOB:EXTRUDE
MOVL C00015 V=30.0 PL=1
CALL JOB:EXTRUDE
MOVL C00016 V=30.0 PL=1
CALL JOB:EXTRUDE
MOVL C00017 V=30.0 PL=1
CALL JOB:EXTRUDE
MOVL C00018 V=30.0 PL=1
CALL JOB:EXTRUDE
MOVL C00019 V=30.0 PL=1
MOVL C00020 V=130.0 PL=1
CALL JOB:EXTRUDE
MOVL C00021 V=30.0 PL=1
CALL JOB:EXTRUDE
MOVL C00022 V=30.0 PL=1
CALL JOB:EXTRUDE
CALL JOB:EXTRUDE
MOVL C00023 V=130.0 PL=1
CALL JOB:EXTRUDE
CALL JOB:EXTRUDE
MOVL C00024 V=30.0 PL=1
CALL JOB:EXTRUDE
MOVL C00025 V=30.0 PL=1
CALL JOB:EXTRUDE
MOVL C00026 V=30.0 PL=1
CALL JOB:EXTRUDE
MOVL C00027 V=30.0 PL=1
MOVL C00028 V=130.0 PL=1
CALL JOB:EXTRUDE
MOVL C00029 V=30.0 PL=1
CALL JOB:EXTRUDE
MOVL C00030 V=30.0 PL=1
CALL JOB:EXTRUDE
MOVL C00031 V=30.0 PL=1
CALL JOB:EXTRUDE
MOVL C00032 V=30.0 PL=1
CALL JOB:EXTRUDE
CALL JOB:EXTRUDE
MOVL C00033 V=130.0 PL=1
CALL JOB:EXTRUDE
CALL JOB:EXTRUDE
MOVL C00034 V=30.0 PL=1
CALL JOB:EXTRUDE
MOVL C00035 V=30.0 PL=1
CALL JOB:EXTRUDE
MOVL C00036 V=30.0 PL=1
CALL JOB:EXTRUDE
MOVL C00037 V=30.0 PL=1
MOVL C00038 V=130.0 PL=1
CALL JOB:EXTRUDE
MOVL C00039 V=30.0 PL=1
MOVL C00040 V=130.0 PL=1
CALL JOB:EXTRUDE
MOVL C00041 V=30.0 PL=1
CALL JOB:EXTRUDE
MOVL C00042 V=30.0 PL=1
MOVL C00043 V=130.0 PL=1
CALL JOB:EXTRUDE
MOVL C00044 V=30.0 PL=1
CALL JOB:EXTRUDE
CALL JOB:EXTRUDE
MOVL C00045 V=130.0 PL=1
CALL JOB:EXTRUDE
CALL JOB:EXTRUDE
MOVL C00046 V=30.0 PL=1
CALL JOB:EXTRUDE
MOVL C00047 V=30.0 PL=1
CALL JOB:EXTRUDE
MOVL C00048 V=30.0 PL=1
CALL JOB:EXTRUDE
MOVL C00049 V=30.0 PL=1
CALL JOB:EXTRUDE
MOVL C00050 V=30.0 PL=1
CALL JOB:EXTRUDE
MOVL C00051 V=30.0 PL=1
MOVL C00052 V=130.0 PL=1
CALL JOB:EXTRUDE
MOVL C00053 V=30.0 PL=1
CALL JOB:EXTRUDE
MOVL C00054 V=30.0 PL=1
MOVL C00055 V=130.0 PL=1
CALL JOB:EXTRUDE
MOVL C00056 V=30.0 PL=1
CALL JOB:EXTRUDE
CALL JOB:EXTRUDE
MOVL C00057 V=130.0 PL=1
CALL JOB:EXTRUDE
CALL JOB:EXTRUDE
MOVL C00058 V=30.0 PL=1
CALL JOB:EXTRUDE
MOVL C00059 V=30.0 PL=1
CALL JOB:EXTRUDE
MOVL C00060 V=30.0 PL=1
CALL JOB:EXTRUDE
MOVL C00061 V=30.0 PL=1
CALL JOB:EXTRUDE
MOVL C00062 V=30.0 PL=1
CALL JOB:EXTRUDE
MOVL C00063 V=30.0 PL=1
CALL JOB:EXTRUDE
MOVL C00064 V=30.0 PL=1
CALL JOB:EXTRUDE
MOVL C00065 V=30.0 PL=1
CALL JOB:EXTRUDE
MOVL C00066 V=30.0 PL=1
MOVL C00067 V=130.0 PL=1
CALL JOB:EXTRUDE
MOVL C00068 V=30.0 PL=1
CALL JOB:EXTRUDE
MOVL C00069 V=30.0 PL=1
CALL JOB:EXTRUDE
MOVL C00070 V=30.0 PL=1
CALL JOB:EXTRUDE
MOVL C00071 V=30.0 PL=1
CALL JOB:EXTRUDE
MOVL C00072 V=30.0 PL=1
CALL JOB:EXTRUDE
MOVL C00073 V=30.0 PL=1
CALL JOB:EXTRUDE
MOVL C00074 V=30.0 PL=1
CALL JOB:EXTRUDE
MOVL C00075 V=30.0 PL=1
CALL JOB:EXTRUDE
MOVL C00076 V=30.0 PL=1
CALL JOB:EXTRUDE
CALL JOB:EXTRUDE
MOVL C00077 V=130.0 PL=1
CALL JOB:EXTRUDE
CALL JOB:EXTRUDE
MOVL C00078 V=30.0 PL=1
CALL JOB:EXTRUDE
MOVL C00079 V=30.0 PL=1
CALL JOB:EXTRUDE
MOVL C00080 V=30.0 PL=1
CALL JOB:EXTRUDE
MOVL C00081 V=30.0 PL=1
CALL JOB:EXTRUDE
MOVL C00082 V=30.0 PL=1
CALL JOB:EXTRUDE
MOVL C00083 V=30.0 PL=1
CALL JOB:EXTRUDE
MOVL C00084 V=30.0 PL=1
CALL JOB:EXTRUDE
MOVL C00085 V=30.0 PL=1
CALL JOB:EXTRUDE
MOVL C00086 V=30.0 PL=1
MOVL C00087 V=130.0 PL=1
CALL JOB:EXTRUDE
MOVL C00088 V=30.0 PL=1
CALL JOB:EXTRUDE
MOVL C00089 V=30.0 PL=1
CALL JOB:EXTRUDE
MOVL C00090 V=30.0 PL=1
CALL JOB:EXTRUDE
MOVL C00091 V=30.0 PL=1
CALL JOB:EXTRUDE
MOVL C00092 V=30.0 PL=1
CALL JOB:EXTRUDE
MOVL C00093 V=30.0 PL=1
CALL JOB:EXTRUDE
MOVL C00094 V=30.0 PL=1
CALL JOB:EXTRUDE
MOVL C00095 V=30.0 PL=1
CALL JOB:EXTRUDE
MOVL C00096 V=30.0 PL=1
CALL JOB:EXTRUDE
CALL JOB:EXTRUDE
MOVL C00097 V=130.0 PL=1
CALL JOB:EXTRUDE
CALL JOB:EXTRUDE
MOVL C00098 V=30.0 PL=1
MOVL C00099 V=130.0 PL=1
CALL JOB:EXTRUDE
MOVL C00100 V=30.0 PL=1
CALL JOB:EXTRUDE
MOVL C00101 V=30.0 PL=1
CALL JOB:EXTRUDE
MOVL C00102 V=30.0 PL=1
CALL JOB:EXTRUDE
MOVL C00103 V=30.0 PL=1
CALL JOB:EXTRUDE
MOVL C00104 V=30.0 PL=1
CALL JOB:EXTRUDE
MOVL C00105 V=30.0 PL=1
MOVL C00106 V=130.0 PL=1
CALL JOB:EXTRUDE
MOVL C00107 V=30.0 PL=1
MOVL C00108 V=130.0 PL=1
CALL JOB:EXTRUDE
MOVL C00109 V=30.0 PL=1
MOVL C00110 V=130.0 PL=1
CALL JOB:EXTRUDE
MOVL C00111 V=30.0 PL=1
CALL JOB:SETRPM(
CALL JOB:MCODEHA
MOVL C00112 V=130.0 PL=1
CALL JOB:EXTRUDE
CALL JOB:EXTRUDE
MOVL C00113 V=130.0 PL=1
CALL JOB:EXTRUDE
CALL JOB:EXTRUDE
MOVL C00114 V=60.0 PL=1
CALL JOB:EXTRUDE
MOVL C00115 V=60.0 PL=1
CALL JOB:EXTRUDE
MOVL C00116 V=60.0 PL=1
CALL JOB:EXTRUDE
MOVL C00117 V=60.0 PL=1
CALL JOB:EXTRUDE
MOVL C00118 V=60.0 PL=1
CALL JOB:EXTRUDE
MOVL C00119 V=60.0 PL=1
CALL JOB:EXTRUDE
MOVL C00120 V=60.0 PL=1
CALL JOB:EXTRUDE
MOVL C00121 V=60.0 PL=1
CALL JOB:EXTRUDE
MOVL C00122 V=60.0 PL=1
CALL JOB:EXTRUDE
MOVL C00123 V=60.0 PL=1
CALL JOB:EXTRUDE
MOVL C00124 V=60.0 PL=1
CALL JOB:EXTRUDE
MOVL C00125 V=60.0 PL=1
CALL JOB:EXTRUDE
MOVL C00126 V=60.0 PL=1
CALL JOB:EXTRUDE
MOVL C00127 V=60.0 PL=1
CALL JOB:EXTRUDE
MOVL C00128 V=60.0 PL=1
CALL JOB:EXTRUDE
MOVL C00129 V=60.0 PL=1
CALL JOB:EXTRUDE
MOVL C00130 V=60.0 PL=1
CALL JOB:EXTRUDE
MOVL C00131 V=60.0 PL=1
CALL JOB:EXTRUDE
MOVL C00132 V=60.0 PL=1
CALL JOB:EXTRUDE
MOVL C00133 V=60.0 PL=1
CALL JOB:EXTRUDE
MOVL C00134 V=60.0 PL=1
CALL JOB:EXTRUDE
MOVL C00135 V=60.0 PL=1
CALL JOB:EXTRUDE
MOVL C00136 V=60.0 PL=1
CALL JOB:EXTRUDE
MOVL C00137 V=60.0 PL=1
CALL JOB:EXTRUDE
MOVL C00138 V=60.0 PL=1
CALL JOB:EXTRUDE
MOVL C00139 V=60.0 PL=1
CALL JOB:EXTRUDE
MOVL C00140 V=60.0 PL=1
CALL JOB:EXTRUDE
MOVL C00141 V=60.0 PL=1
CALL JOB:EXTRUDE
MOVL C00142 V=60.0 PL=1
CALL JOB:EXTRUDE
MOVL C00143 V=60.0 PL=1
MOVL C00144 V=130.0 PL=1
CALL JOB:EXTRUDE
MOVL C00145 V=60.0 PL=1
CALL JOB:EXTRUDE
MOVL C00146 V=60.0 PL=1
CALL JOB:EXTRUDE
MOVL C00147 V=60.0 PL=1
CALL JOB:EXTRUDE
MOVL C00148 V=60.0 PL=1
CALL JOB:EXTRUDE
MOVL C00149 V=60.0 PL=1
CALL JOB:EXTRUDE
MOVL C00150 V=60.0 PL=1
CALL JOB:EXTRUDE
MOVL C00151 V=60.0 PL=1
CALL JOB:EXTRUDE
MOVL C00152 V=60.0 PL=1
CALL JOB:EXTRUDE
MOVL C00153 V=60.0 PL=1
CALL JOB:EXTRUDE
MOVL C00154 V=60.0 PL=1
CALL JOB:EXTRUDE
MOVL C00155 V=60.0 PL=1
CALL JOB:EXTRUDE
MOVL C00156 V=60.0 PL=1
CALL JOB:EXTRUDE
MOVL C00157 V=60.0 PL=1
CALL JOB:EXTRUDE
MOVL C00158 V=60.0 PL=1
CALL JOB:EXTRUDE
MOVL C00159 V=60.0 PL=1
CALL JOB:EXTRUDE
MOVL C00160 V=60.0 PL=1
CALL JOB:EXTRUDE
MOVL C00161 V=60.0 PL=1
CALL JOB:EXTRUDE
MOVL C00162 V=60.0 PL=1
CALL JOB:EXTRUDE
MOVL C00163 V=60.0 PL=1
CALL JOB:EXTRUDE
MOVL C00164 V=60.0 PL=1
CALL JOB:EXTRUDE
MOVL C00165 V=60.0 PL=1
CALL JOB:EXTRUDE
MOVL C00166 V=60.0 PL=1
CALL JOB:EXTRUDE
MOVL C00167 V=60.0 PL=1
CALL JOB:EXTRUDE
MOVL C00168 V=60.0 PL=1
CALL JOB:EXTRUDE
MOVL C00169 V=60.0 PL=1
CALL JOB:EXTRUDE
MOVL C00170 V=60.0 PL=1
CALL JOB:EXTRUDE
MOVL C00171 V=60.0 PL=1
CALL JOB:EXTRUDE
MOVL C00172 V=60.0 PL=1
CALL JOB:EXTRUDE
MOVL C00173 V=60.0 PL=1
CALL JOB:EXTRUDE
MOVL C00174 V=60.0 PL=1
CALL JOB:EXTRUDE
MOVL C00175 V=60.0 PL=1
CALL JOB:EXTRUDE
MOVL C00176 V=60.0 PL=1
CALL JOB:EXTRUDE
MOVL C00177 V=60.0 PL=1
CALL JOB:EXTRUDE
MOVL C00178 V=60.0 PL=1
CALL JOB:EXTRUDE
MOVL C00179 V=60.0 PL=1
CALL JOB:EXTRUDE
MOVL C00180 V=60.0 PL=1
CALL JOB:EXTRUDE
MOVL C00181 V=60.0 PL=1
CALL JOB:EXTRUDE
MOVL C00182 V=60.0 PL=1
CALL JOB:EXTRUDE
MOVL C00183 V=60.0 PL=1
CALL JOB:EXTRUDE
MOVL C00184 V=60.0 PL=1
CALL JOB:EXTRUDE
MOVL C00185 V=60.0 PL=1
CALL JOB:EXTRUDE
MOVL C00186 V=60.0 PL=1
MOVL C00187 V=130.0 PL=1
CALL JOB:EXTRUDE
MOVL C00188 V=30.0 PL=1
CALL JOB:EXTRUDE
MOVL C00189 V=30.0 PL=1
CALL JOB:EXTRUDE
MOVL C00190 V=30.0 PL=1
CALL JOB:EXTRUDE
MOVL C00191 V=30.0 PL=1
CALL JOB:EXTRUDE
MOVL C00192 V=30.0 PL=1
CALL JOB:EXTRUDE
MOVL C00193 V=30.0 PL=1
CALL JOB:EXTRUDE
MOVL C00194 V=30.0 PL=1
CALL JOB:EXTRUDE
MOVL C00195 V=30.0 PL=1
CALL JOB:EXTRUDE
MOVL C00196 V=30.0 PL=1
CALL JOB:EXTRUDE
MOVL C00197 V=30.0 PL=1
CALL JOB:EXTRUDE
MOVL C00198 V=30.0 PL=1
CALL JOB:EXTRUDE
MOVL C00199 V=30.0 PL=1
CALL JOB:EXTRUDE
MOVL C00200 V=30.0 PL=1
CALL JOB:EXTRUDE
MOVL C00201 V=30.0 PL=1
CALL JOB:EXTRUDE
MOVL C00202 V=30.0 PL=1
CALL JOB:EXTRUDE
MOVL C00203 V=30.0 PL=1
CALL JOB:EXTRUDE
MOVL C00204 V=30.0 PL=1
CALL JOB:EXTRUDE
MOVL C00205 V=30.0 PL=1
CALL JOB:EXTRUDE
MOVL C00206 V=30.0 PL=1
CALL JOB:EXTRUDE
MOVL C00207 V=30.0 PL=1
CALL JOB:EXTRUDE
MOVL C00208 V=30.0 PL=1
CALL JOB:EXTRUDE
MOVL C00209 V=30.0 PL=1
CALL JOB:EXTRUDE
MOVL C00210 V=30.0 PL=1
CALL JOB:EXTRUDE
MOVL C00211 V=30.0 PL=1
CALL JOB:EXTRUDE
MOVL C00212 V=30.0 PL=1
CALL JOB:EXTRUDE
MOVL C00213 V=30.0 PL=1
CALL JOB:EXTRUDE
MOVL C00214 V=30.0 PL=1
CALL JOB:EXTRUDE
MOVL C00215 V=30.0 PL=1
CALL JOB:EXTRUDE
MOVL C00216 V=30.0 PL=1
CALL JOB:EXTRUDE
MOVL C00217 V=30.0 PL=1
CALL JOB:EXTRUDE
MOVL C00218 V=30.0 PL=1
CALL JOB:EXTRUDE
MOVL C00219 V=30.0 PL=1
CALL JOB:EXTRUDE
MOVL C00220 V=30.0 PL=1
CALL JOB:EXTRUDE
MOVL C00221 V=30.0 PL=1
CALL JOB:EXTRUDE
MOVL C00222 V=30.0 PL=1
CALL JOB:EXTRUDE
MOVL C00223 V=30.0 PL=1
CALL JOB:EXTRUDE
MOVL C00224 V=30.0 PL=1
CALL JOB:EXTRUDE
MOVL C00225 V=30.0 PL=1
CALL JOB:EXTRUDE
MOVL C00226 V=30.0 PL=1
CALL JOB:EXTRUDE
MOVL C00227 V=30.0 PL=1
CALL JOB:EXTRUDE
MOVL C00228 V=30.0 PL=1
CALL JOB:EXTRUDE
MOVL C00229 V=30.0 PL=1
CALL JOB:EXTRUDE
MOVL C00230 V=30.0 PL=1
CALL JOB:EXTRUDE
MOVL C00231 V=30.0 PL=1
CALL JOB:EXTRUDE
MOVL C00232 V=30.0 PL=1
CALL JOB:EXTRUDE
MOVL C00233 V=30.0 PL=1
CALL JOB:EXTRUDE
MOVL C00234 V=30.0 PL=1
CALL JOB:EXTRUDE
MOVL C00235 V=30.0 PL=1
CALL JOB:EXTRUDE
MOVL C00236 V=30.0 PL=1
CALL JOB:EXTRUDE
MOVL C00237 V=30.0 PL=1
CALL JOB:EXTRUDE
MOVL C00238 V=30.0 PL=1
CALL JOB:EXTRUDE
MOVL C00239 V=30.0 PL=1
CALL JOB:EXTRUDE
MOVL C00240 V=30.0 PL=1
CALL JOB:EXTRUDE
MOVL C00241 V=30.0 PL=1
CALL JOB:EXTRUDE
MOVL C00242 V=30.0 PL=1
CALL JOB:EXTRUDE
MOVL C00243 V=30.0 PL=1
CALL JOB:EXTRUDE
MOVL C00244 V=30.0 PL=1
CALL JOB:EXTRUDE
MOVL C00245 V=30.0 PL=1
CALL JOB:EXTRUDE
MOVL C00246 V=30.0 PL=1
CALL JOB:EXTRUDE
MOVL C00247 V=30.0 PL=1
CALL JOB:EXTRUDE
MOVL C00248 V=30.0 PL=1
CALL JOB:EXTRUDE
MOVL C00249 V=30.0 PL=1
CALL JOB:EXTRUDE
MOVL C00250 V=30.0 PL=1
CALL JOB:EXTRUDE
MOVL C00251 V=30.0 PL=1
CALL JOB:EXTRUDE
MOVL C00252 V=30.0 PL=1
CALL JOB:EXTRUDE
MOVL C00253 V=30.0 PL=1
CALL JOB:EXTRUDE
MOVL C00254 V=30.0 PL=1
CALL JOB:EXTRUDE
MOVL C00255 V=30.0 PL=1
CALL JOB:EXTRUDE
MOVL C00256 V=30.0 PL=1
CALL JOB:EXTRUDE
MOVL C00257 V=30.0 PL=1
CALL JOB:EXTRUDE
MOVL C00258 V=30.0 PL=1
CALL JOB:EXTRUDE
MOVL C00259 V=30.0 PL=1
MOVL C00260 V=130.0 PL=1
CALL JOB:EXTRUDE
CALL JOB:EXTRUDE
MOVL C00261 V=130.0 PL=1
CALL JOB:EXTRUDE
CALL JOB:EXTRUDE
MOVL C00262 V=30.0 PL=1
CALL JOB:EXTRUDE
MOVL C00263 V=30.0 PL=1
CALL JOB:EXTRUDE
MOVL C00264 V=30.0 PL=1
CALL JOB:EXTRUDE
MOVL C00265 V=30.0 PL=1
CALL JOB:EXTRUDE
MOVL C00266 V=30.0 PL=1
CALL JOB:EXTRUDE
MOVL C00267 V=30.0 PL=1
CALL JOB:EXTRUDE
MOVL C00268 V=30.0 PL=1
CALL JOB:EXTRUDE
MOVL C00269 V=30.0 PL=1
CALL JOB:EXTRUDE
MOVL C00270 V=30.0 PL=1
CALL JOB:EXTRUDE
MOVL C00271 V=30.0 PL=1
CALL JOB:EXTRUDE
MOVL C00272 V=30.0 PL=1
CALL JOB:EXTRUDE
MOVL C00273 V=30.0 PL=1
CALL JOB:EXTRUDE
MOVL C00274 V=30.0 PL=1
CALL JOB:EXTRUDE
MOVL C00275 V=30.0 PL=1
CALL JOB:EXTRUDE
MOVL C00276 V=30.0 PL=1
CALL JOB:EXTRUDE
MOVL C00277 V=30.0 PL=1
CALL JOB:EXTRUDE
MOVL C00278 V=30.0 PL=1
CALL JOB:EXTRUDE
MOVL C00279 V=30.0 PL=1
CALL JOB:EXTRUDE
MOVL C00280 V=30.0 PL=1
CALL JOB:EXTRUDE
MOVL C00281 V=30.0 PL=1
CALL JOB:EXTRUDE
MOVL C00282 V=30.0 PL=1
CALL JOB:EXTRUDE
MOVL C00283 V=30.0 PL=1
CALL JOB:EXTRUDE
MOVL C00284 V=30.0 PL=1
CALL JOB:EXTRUDE
MOVL C00285 V=30.0 PL=1
CALL JOB:EXTRUDE
MOVL C00286 V=30.0 PL=1
CALL JOB:EXTRUDE
MOVL C00287 V=30.0 PL=1
CALL JOB:EXTRUDE
MOVL C00288 V=30.0 PL=1
CALL JOB:EXTRUDE
MOVL C00289 V=30.0 PL=1
CALL JOB:EXTRUDE
MOVL C00290 V=30.0 PL=1
CALL JOB:EXTRUDE
MOVL C00291 V=30.0 PL=1
CALL JOB:EXTRUDE
MOVL C00292 V=30.0 PL=1
CALL JOB:EXTRUDE
MOVL C00293 V=30.0 PL=1
CALL JOB:EXTRUDE
MOVL C00294 V=30.0 PL=1
CALL JOB:EXTRUDE
MOVL C00295 V=30.0 PL=1
CALL JOB:EXTRUDE
MOVL C00296 V=30.0 PL=1
CALL JOB:EXTRUDE
MOVL C00297 V=30.0 PL=1
CALL JOB:EXTRUDE
MOVL C00298 V=30.0 PL=1
CALL JOB:EXTRUDE
MOVL C00299 V=30.0 PL=1
CALL JOB:EXTRUDE
MOVL C00300 V=30.0 PL=1
CALL JOB:EXTRUDE
MOVL C00301 V=30.0 PL=1
CALL JOB:EXTRUDE
MOVL C00302 V=30.0 PL=1
CALL JOB:EXTRUDE
MOVL C00303 V=30.0 PL=1
CALL JOB:EXTRUDE
MOVL C00304 V=30.0 PL=1
CALL JOB:EXTRUDE
MOVL C00305 V=30.0 PL=1
CALL JOB:EXTRUDE
MOVL C00306 V=30.0 PL=1
CALL JOB:EXTRUDE
MOVL C00307 V=30.0 PL=1
CALL JOB:EXTRUDE
MOVL C00308 V=30.0 PL=1
CALL JOB:EXTRUDE
MOVL C00309 V=30.0 PL=1
CALL JOB:EXTRUDE
MOVL C00310 V=30.0 PL=1
CALL JOB:EXTRUDE
MOVL C00311 V=30.0 PL=1
CALL JOB:EXTRUDE
MOVL C00312 V=30.0 PL=1
CALL JOB:EXTRUDE
MOVL C00313 V=30.0 PL=1
CALL JOB:EXTRUDE
MOVL C00314 V=30.0 PL=1
CALL JOB:EXTRUDE
MOVL C00315 V=30.0 PL=1
CALL JOB:EXTRUDE
MOVL C00316 V=30.0 PL=1
CALL JOB:EXTRUDE
MOVL C00317 V=30.0 PL=1
CALL JOB:EXTRUDE
MOVL C00318 V=30.0 PL=1
CALL JOB:EXTRUDE
MOVL C00319 V=30.0 PL=1
CALL JOB:EXTRUDE
MOVL C00320 V=30.0 PL=1
CALL JOB:EXTRUDE
MOVL C00321 V=30.0 PL=1
CALL JOB:EXTRUDE
MOVL C00322 V=30.0 PL=1
CALL JOB:EXTRUDE
MOVL C00323 V=30.0 PL=1
CALL JOB:EXTRUDE
MOVL C00324 V=30.0 PL=1
CALL JOB:EXTRUDE
MOVL C00325 V=30.0 PL=1
CALL JOB:EXTRUDE
MOVL C00326 V=30.0 PL=1
CALL JOB:EXTRUDE
MOVL C00327 V=30.0 PL=1
CALL JOB:EXTRUDE
MOVL C00328 V=30.0 PL=1
CALL JOB:EXTRUDE
MOVL C00329 V=30.0 PL=1
CALL JOB:EXTRUDE
MOVL C00330 V=30.0 PL=1
CALL JOB:EXTRUDE
MOVL C00331 V=30.0 PL=1
CALL JOB:EXTRUDE
MOVL C00332 V=30.0 PL=1
CALL JOB:EXTRUDE
MOVL C00333 V=30.0 PL=1
CALL JOB:EXTRUDE
MOVL C00334 V=30.0 PL=1
CALL JOB:EXTRUDE
MOVL C00335 V=30.0 PL=1
CALL JOB:EXTRUDE
MOVL C00336 V=30.0 PL=1
CALL JOB:EXTRUDE
MOVL C00337 V=30.0 PL=1
CALL JOB:EXTRUDE
MOVL C00338 V=30.0 PL=1
CALL JOB:EXTRUDE
MOVL C00339 V=30.0 PL=1
CALL JOB:EXTRUDE
MOVL C00340 V=30.0 PL=1
CALL JOB:EXTRUDE
MOVL C00341 V=30.0 PL=1
CALL JOB:EXTRUDE
MOVL C00342 V=30.0 PL=1
CALL JOB:EXTRUDE
MOVL C00343 V=30.0 PL=1
CALL JOB:EXTRUDE
MOVL C00344 V=30.0 PL=1
CALL JOB:EXTRUDE
MOVL C00345 V=30.0 PL=1
CALL JOB:EXTRUDE
MOVL C00346 V=30.0 PL=1
CALL JOB:EXTRUDE
MOVL C00347 V=30.0 PL=1
CALL JOB:EXTRUDE
MOVL C00348 V=30.0 PL=1
CALL JOB:EXTRUDE
MOVL C00349 V=30.0 PL=1
CALL JOB:EXTRUDE
MOVL C00350 V=30.0 PL=1
CALL JOB:EXTRUDE
MOVL C00351 V=30.0 PL=1
CALL JOB:EXTRUDE
MOVL C00352 V=30.0 PL=1
CALL JOB:EXTRUDE
MOVL C00353 V=30.0 PL=1
CALL JOB:EXTRUDE
MOVL C00354 V=30.0 PL=1
MOVL C00355 V=130.0 PL=1
CALL JOB:EXTRUDE
MOVL C00356 V=30.0 PL=1
CALL JOB:EXTRUDE
MOVL C00357 V=30.0 PL=1
CALL JOB:EXTRUDE
MOVL C00358 V=30.0 PL=1
CALL JOB:EXTRUDE
MOVL C00359 V=30.0 PL=1
CALL JOB:EXTRUDE
MOVL C00360 V=30.0 PL=1
CALL JOB:EXTRUDE
MOVL C00361 V=30.0 PL=1
CALL JOB:EXTRUDE
MOVL C00362 V=30.0 PL=1
CALL JOB:EXTRUDE
MOVL C00363 V=30.0 PL=1
CALL JOB:EXTRUDE
MOVL C00364 V=30.0 PL=1
CALL JOB:EXTRUDE
MOVL C00365 V=30.0 PL=1
CALL JOB:EXTRUDE
MOVL C00366 V=30.0 PL=1
CALL JOB:EXTRUDE
MOVL C00367 V=30.0 PL=1
CALL JOB:EXTRUDE
MOVL C00368 V=30.0 PL=1
CALL JOB:EXTRUDE
MOVL C00369 V=30.0 PL=1
CALL JOB:EXTRUDE
MOVL C00370 V=30.0 PL=1
CALL JOB:EXTRUDE
MOVL C00371 V=30.0 PL=1
CALL JOB:EXTRUDE
MOVL C00372 V=30.0 PL=1
CALL JOB:EXTRUDE
MOVL C00373 V=30.0 PL=1
CALL JOB:EXTRUDE
MOVL C00374 V=30.0 PL=1
CALL JOB:EXTRUDE
MOVL C00375 V=30.0 PL=1
CALL JOB:EXTRUDE
MOVL C00376 V=30.0 PL=1
CALL JOB:EXTRUDE
MOVL C00377 V=30.0 PL=1
CALL JOB:EXTRUDE
MOVL C00378 V=30.0 PL=1
CALL JOB:EXTRUDE
MOVL C00379 V=30.0 PL=1
CALL JOB:EXTRUDE
MOVL C00380 V=30.0 PL=1
CALL JOB:EXTRUDE
MOVL C00381 V=30.0 PL=1
CALL JOB:EXTRUDE
MOVL C00382 V=30.0 PL=1
CALL JOB:EXTRUDE
MOVL C00383 V=30.0 PL=1
CALL JOB:EXTRUDE
MOVL C00384 V=30.0 PL=1
CALL JOB:EXTRUDE
MOVL C00385 V=30.0 PL=1
CALL JOB:EXTRUDE
MOVL C00386 V=30.0 PL=1
CALL JOB:EXTRUDE
MOVL C00387 V=30.0 PL=1
CALL JOB:EXTRUDE
MOVL C00388 V=30.0 PL=1
CALL JOB:EXTRUDE
MOVL C00389 V=30.0 PL=1
CALL JOB:EXTRUDE
MOVL C00390 V=30.0 PL=1
CALL JOB:EXTRUDE
MOVL C00391 V=30.0 PL=1
CALL JOB:EXTRUDE
MOVL C00392 V=30.0 PL=1
CALL JOB:EXTRUDE
MOVL C00393 V=30.0 PL=1
CALL JOB:EXTRUDE
MOVL C00394 V=30.0 PL=1
CALL JOB:EXTRUDE
MOVL C00395 V=30.0 PL=1
CALL JOB:EXTRUDE
MOVL C00396 V=30.0 PL=1
CALL JOB:EXTRUDE
MOVL C00397 V=30.0 PL=1
CALL JOB:EXTRUDE
MOVL C00398 V=30.0 PL=1
CALL JOB:EXTRUDE
MOVL C00399 V=30.0 PL=1
CALL JOB:EXTRUDE
MOVL C00400 V=30.0 PL=1
CALL JOB:EXTRUDE
MOVL C00401 V=30.0 PL=1
CALL JOB:EXTRUDE
MOVL C00402 V=30.0 PL=1
CALL JOB:EXTRUDE
MOVL C00403 V=30.0 PL=1
CALL JOB:EXTRUDE
MOVL C00404 V=30.0 PL=1
CALL JOB:EXTRUDE
MOVL C00405 V=30.0 PL=1
CALL JOB:EXTRUDE
MOVL C00406 V=30.0 PL=1
CALL JOB:EXTRUDE
MOVL C00407 V=30.0 PL=1
CALL JOB:EXTRUDE
MOVL C00408 V=30.0 PL=1
CALL JOB:EXTRUDE
MOVL C00409 V=30.0 PL=1
CALL JOB:EXTRUDE
MOVL C00410 V=30.0 PL=1
CALL JOB:EXTRUDE
MOVL C00411 V=30.0 PL=1
CALL JOB:EXTRUDE
MOVL C00412 V=30.0 PL=1
CALL JOB:EXTRUDE
MOVL C00413 V=30.0 PL=1
CALL JOB:EXTRUDE
MOVL C00414 V=30.0 PL=1
CALL JOB:EXTRUDE
MOVL C00415 V=30.0 PL=1
CALL JOB:EXTRUDE
MOVL C00416 V=30.0 PL=1
CALL JOB:EXTRUDE
MOVL C00417 V=30.0 PL=1
CALL JOB:EXTRUDE
MOVL C00418 V=30.0 PL=1
CALL JOB:EXTRUDE
MOVL C00419 V=30.0 PL=1
CALL JOB:EXTRUDE
MOVL C00420 V=30.0 PL=1
CALL JOB:EXTRUDE
MOVL C00421 V=30.0 PL=1
CALL JOB:EXTRUDE
MOVL C00422 V=30.0 PL=1
CALL JOB:EXTRUDE
MOVL C00423 V=30.0 PL=1
CALL JOB:EXTRUDE
MOVL C00424 V=30.0 PL=1
CALL JOB:EXTRUDE
MOVL C00425 V=30.0 PL=1
CALL JOB:EXTRUDE
MOVL C00426 V=30.0 PL=1
CALL JOB:EXTRUDE
MOVL C00427 V=30.0 PL=1
CALL JOB:EXTRUDE
MOVL C00428 V=30.0 PL=1
CALL JOB:EXTRUDE
MOVL C00429 V=30.0 PL=1
CALL JOB:EXTRUDE
MOVL C00430 V=30.0 PL=1
CALL JOB:EXTRUDE
MOVL C00431 V=30.0 PL=1
CALL JOB:EXTRUDE
MOVL C00432 V=30.0 PL=1
CALL JOB:EXTRUDE
MOVL C00433 V=30.0 PL=1
CALL JOB:EXTRUDE
MOVL C00434 V=30.0 PL=1
CALL JOB:EXTRUDE
MOVL C00435 V=30.0 PL=1
CALL JOB:EXTRUDE
MOVL C00436 V=30.0 PL=1
CALL JOB:EXTRUDE
MOVL C00437 V=30.0 PL=1
CALL JOB:EXTRUDE
MOVL C00438 V=30.0 PL=1
CALL JOB:EXTRUDE
MOVL C00439 V=30.0 PL=1
CALL JOB:EXTRUDE
MOVL C00440 V=30.0 PL=1
CALL JOB:EXTRUDE
MOVL C00441 V=30.0 PL=1
CALL JOB:EXTRUDE
MOVL C00442 V=30.0 PL=1
CALL JOB:EXTRUDE
MOVL C00443 V=30.0 PL=1
CALL JOB:EXTRUDE
MOVL C00444 V=30.0 PL=1
CALL JOB:EXTRUDE
MOVL C00445 V=30.0 PL=1
CALL JOB:EXTRUDE
MOVL C00446 V=30.0 PL=1
CALL JOB:EXTRUDE
MOVL C00447 V=30.0 PL=1
CALL JOB:EXTRUDE
MOVL C00448 V=30.0 PL=1
CALL JOB:EXTRUDE
MOVL C00449 V=30.0 PL=1
CALL JOB:EXTRUDE
CALL JOB:EXTRUDE
MOVL C00450 V=130.0 PL=1
CALL JOB:EXTRUDE
CALL JOB:EXTRUDE
MOVL C00451 V=30.0 PL=1
CALL JOB:EXTRUDE
MOVL C00452 V=30.0 PL=1
CALL JOB:EXTRUDE
MOVL C00453 V=30.0 PL=1
CALL JOB:EXTRUDE
MOVL C00454 V=30.0 PL=1
CALL JOB:EXTRUDE
MOVL C00455 V=30.0 PL=1
CALL JOB:EXTRUDE
MOVL C00456 V=30.0 PL=1
CALL JOB:EXTRUDE
MOVL C00457 V=30.0 PL=1
CALL JOB:EXTRUDE
MOVL C00458 V=30.0 PL=1
CALL JOB:EXTRUDE
MOVL C00459 V=30.0 PL=1
CALL JOB:EXTRUDE
MOVL C00460 V=30.0 PL=1
CALL JOB:EXTRUDE
MOVL C00461 V=30.0 PL=1
CALL JOB:EXTRUDE
MOVL C00462 V=30.0 PL=1
CALL JOB:EXTRUDE
MOVL C00463 V=30.0 PL=1
CALL JOB:EXTRUDE
MOVL C00464 V=30.0 PL=1
CALL JOB:EXTRUDE
MOVL C00465 V=30.0 PL=1
CALL JOB:EXTRUDE
MOVL C00466 V=30.0 PL=1
CALL JOB:EXTRUDE
MOVL C00467 V=30.0 PL=1
CALL JOB:EXTRUDE
MOVL C00468 V=30.0 PL=1
CALL JOB:EXTRUDE
MOVL C00469 V=30.0 PL=1
CALL JOB:EXTRUDE
MOVL C00470 V=30.0 PL=1
CALL JOB:EXTRUDE
MOVL C00471 V=30.0 PL=1
CALL JOB:EXTRUDE
MOVL C00472 V=30.0 PL=1
CALL JOB:EXTRUDE
MOVL C00473 V=30.0 PL=1
CALL JOB:EXTRUDE
MOVL C00474 V=30.0 PL=1
CALL JOB:EXTRUDE
MOVL C00475 V=30.0 PL=1
CALL JOB:EXTRUDE
MOVL C00476 V=30.0 PL=1
CALL JOB:EXTRUDE
MOVL C00477 V=30.0 PL=1
CALL JOB:EXTRUDE
MOVL C00478 V=30.0 PL=1
CALL JOB:EXTRUDE
MOVL C00479 V=30.0 PL=1
CALL JOB:EXTRUDE
MOVL C00480 V=30.0 PL=1
CALL JOB:EXTRUDE
MOVL C00481 V=30.0 PL=1
CALL JOB:EXTRUDE
MOVL C00482 V=30.0 PL=1
CALL JOB:EXTRUDE
MOVL C00483 V=30.0 PL=1
CALL JOB:EXTRUDE
MOVL C00484 V=30.0 PL=1
CALL JOB:EXTRUDE
MOVL C00485 V=30.0 PL=1
CALL JOB:EXTRUDE
MOVL C00486 V=30.0 PL=1
CALL JOB:EXTRUDE
MOVL C00487 V=30.0 PL=1
CALL JOB:EXTRUDE
MOVL C00488 V=30.0 PL=1
CALL JOB:EXTRUDE
MOVL C00489 V=30.0 PL=1
CALL JOB:EXTRUDE
MOVL C00490 V=30.0 PL=1
CALL JOB:EXTRUDE
MOVL C00491 V=30.0 PL=1
CALL JOB:EXTRUDE
MOVL C00492 V=30.0 PL=1
CALL JOB:EXTRUDE
MOVL C00493 V=30.0 PL=1
CALL JOB:EXTRUDE
MOVL C00494 V=30.0 PL=1
CALL JOB:EXTRUDE
MOVL C00495 V=30.0 PL=1
CALL JOB:EXTRUDE
MOVL C00496 V=30.0 PL=1
CALL JOB:EXTRUDE
MOVL C00497 V=30.0 PL=1
CALL JOB:EXTRUDE
MOVL C00498 V=30.0 PL=1
CALL JOB:EXTRUDE
MOVL C00499 V=30.0 PL=1
CALL JOB:EXTRUDE
MOVL C00500 V=30.0 PL=1
CALL JOB:EXTRUDE
MOVL C00501 V=30.0 PL=1
CALL JOB:EXTRUDE
MOVL C00502 V=30.0 PL=1
CALL JOB:EXTRUDE
MOVL C00503 V=30.0 PL=1
CALL JOB:EXTRUDE
MOVL C00504 V=30.0 PL=1
CALL JOB:EXTRUDE
MOVL C00505 V=30.0 PL=1
CALL JOB:EXTRUDE
MOVL C00506 V=30.0 PL=1
CALL JOB:EXTRUDE
MOVL C00507 V=30.0 PL=1
CALL JOB:EXTRUDE
MOVL C00508 V=30.0 PL=1
CALL JOB:EXTRUDE
MOVL C00509 V=30.0 PL=1
CALL JOB:EXTRUDE
MOVL C00510 V=30.0 PL=1
CALL JOB:EXTRUDE
MOVL C00511 V=30.0 PL=1
CALL JOB:EXTRUDE
MOVL C00512 V=30.0 PL=1
CALL JOB:EXTRUDE
MOVL C00513 V=30.0 PL=1
CALL JOB:EXTRUDE
MOVL C00514 V=30.0 PL=1
CALL JOB:EXTRUDE
MOVL C00515 V=30.0 PL=1
CALL JOB:EXTRUDE
MOVL C00516 V=30.0 PL=1
CALL JOB:EXTRUDE
MOVL C00517 V=30.0 PL=1
CALL JOB:EXTRUDE
MOVL C00518 V=30.0 PL=1
CALL JOB:EXTRUDE
MOVL C00519 V=30.0 PL=1
CALL JOB:EXTRUDE
MOVL C00520 V=30.0 PL=1
CALL JOB:EXTRUDE
MOVL C00521 V=30.0 PL=1
CALL JOB:EXTRUDE
MOVL C00522 V=30.0 PL=1
CALL JOB:EXTRUDE
MOVL C00523 V=30.0 PL=1
CALL JOB:EXTRUDE
MOVL C00524 V=30.0 PL=1
CALL JOB:EXTRUDE
MOVL C00525 V=30.0 PL=1
CALL JOB:EXTRUDE
MOVL C00526 V=30.0 PL=1
CALL JOB:EXTRUDE
MOVL C00527 V=30.0 PL=1
CALL JOB:EXTRUDE
MOVL C00528 V=30.0 PL=1
CALL JOB:EXTRUDE
MOVL C00529 V=30.0 PL=1
CALL JOB:EXTRUDE
MOVL C00530 V=30.0 PL=1
CALL JOB:EXTRUDE
MOVL C00531 V=30.0 PL=1
CALL JOB:EXTRUDE
MOVL C00532 V=30.0 PL=1
CALL JOB:EXTRUDE
MOVL C00533 V=30.0 PL=1
CALL JOB:EXTRUDE
MOVL C00534 V=30.0 PL=1
CALL JOB:EXTRUDE
MOVL C00535 V=30.0 PL=1
CALL JOB:EXTRUDE
MOVL C00536 V=30.0 PL=1
CALL JOB:EXTRUDE
MOVL C00537 V=30.0 PL=1
CALL JOB:EXTRUDE
MOVL C00538 V=30.0 PL=1
CALL JOB:EXTRUDE
MOVL C00539 V=30.0 PL=1
CALL JOB:EXTRUDE
MOVL C00540 V=30.0 PL=1
CALL JOB:EXTRUDE
MOVL C00541 V=30.0 PL=1
CALL JOB:EXTRUDE
MOVL C00542 V=30.0 PL=1
CALL JOB:EXTRUDE
MOVL C00543 V=30.0 PL=1
CALL JOB:EXTRUDE
MOVL C00544 V=30.0 PL=1
CALL JOB:EXTRUDE
MOVL C00545 V=30.0 PL=1
CALL JOB:EXTRUDE
MOVL C00546 V=30.0 PL=1
CALL JOB:EXTRUDE
MOVL C00547 V=30.0 PL=1
CALL JOB:EXTRUDE
MOVL C00548 V=30.0 PL=1
CALL JOB:EXTRUDE
MOVL C00549 V=30.0 PL=1
CALL JOB:EXTRUDE
MOVL C00550 V=30.0 PL=1
CALL JOB:EXTRUDE
MOVL C00551 V=30.0 PL=1
CALL JOB:EXTRUDE
MOVL C00552 V=30.0 PL=1
CALL JOB:EXTRUDE
MOVL C00553 V=30.0 PL=1
CALL JOB:EXTRUDE
MOVL C00554 V=30.0 PL=1
CALL JOB:EXTRUDE
MOVL C00555 V=30.0 PL=1
CALL JOB:EXTRUDE
MOVL C00556 V=30.0 PL=1
CALL JOB:EXTRUDE
MOVL C00557 V=30.0 PL=1
CALL JOB:EXTRUDE
MOVL C00558 V=30.0 PL=1
CALL JOB:EXTRUDE
MOVL C00559 V=30.0 PL=1
CALL JOB:EXTRUDE
MOVL C00560 V=30.0 PL=1
CALL JOB:EXTRUDE
MOVL C00561 V=30.0 PL=1
CALL JOB:EXTRUDE
MOVL C00562 V=30.0 PL=1
CALL JOB:EXTRUDE
MOVL C00563 V=30.0 PL=1
CALL JOB:EXTRUDE
MOVL C00564 V=30.0 PL=1
CALL JOB:EXTRUDE
MOVL C00565 V=30.0 PL=1
CALL JOB:EXTRUDE
MOVL C00566 V=30.0 PL=1
CALL JOB:EXTRUDE
MOVL C00567 V=30.0 PL=1
CALL JOB:EXTRUDE
MOVL C00568 V=30.0 PL=1
CALL JOB:EXTRUDE
MOVL C00569 V=30.0 PL=1
CALL JOB:EXTRUDE
MOVL C00570 V=30.0 PL=1
CALL JOB:EXTRUDE
MOVL C00571 V=30.0 PL=1
CALL JOB:EXTRUDE
MOVL C00572 V=30.0 PL=1
CALL JOB:EXTRUDE
CALL JOB:EXTRUDE
MOVL C00573 V=130.0 PL=1
CALL JOB:EXTRUDE
CALL JOB:EXTRUDE
MOVL C00574 V=30.0 PL=1
CALL JOB:EXTRUDE
MOVL C00575 V=30.0 PL=1
CALL JOB:EXTRUDE
MOVL C00576 V=30.0 PL=1
CALL JOB:EXTRUDE
MOVL C00577 V=30.0 PL=1
CALL JOB:EXTRUDE
MOVL C00578 V=30.0 PL=1
CALL JOB:EXTRUDE
MOVL C00579 V=30.0 PL=1
CALL JOB:EXTRUDE
MOVL C00580 V=30.0 PL=1
CALL JOB:EXTRUDE
MOVL C00581 V=30.0 PL=1
CALL JOB:EXTRUDE
MOVL C00582 V=30.0 PL=1
CALL JOB:EXTRUDE
MOVL C00583 V=30.0 PL=1
CALL JOB:EXTRUDE
MOVL C00584 V=30.0 PL=1
CALL JOB:EXTRUDE
MOVL C00585 V=30.0 PL=1
CALL JOB:EXTRUDE
MOVL C00586 V=30.0 PL=1
CALL JOB:EXTRUDE
MOVL C00587 V=30.0 PL=1
CALL JOB:EXTRUDE
MOVL C00588 V=30.0 PL=1
CALL JOB:EXTRUDE
MOVL C00589 V=30.0 PL=1
CALL JOB:EXTRUDE
MOVL C00590 V=30.0 PL=1
CALL JOB:EXTRUDE
MOVL C00591 V=30.0 PL=1
CALL JOB:EXTRUDE
MOVL C00592 V=30.0 PL=1
CALL JOB:EXTRUDE
MOVL C00593 V=30.0 PL=1
CALL JOB:EXTRUDE
MOVL C00594 V=30.0 PL=1
CALL JOB:EXTRUDE
MOVL C00595 V=30.0 PL=1
CALL JOB:EXTRUDE
MOVL C00596 V=30.0 PL=1
CALL JOB:EXTRUDE
MOVL C00597 V=30.0 PL=1
CALL JOB:EXTRUDE
MOVL C00598 V=30.0 PL=1
CALL JOB:EXTRUDE
MOVL C00599 V=30.0 PL=1
CALL JOB:EXTRUDE
MOVL C00600 V=30.0 PL=1
CALL JOB:EXTRUDE
MOVL C00601 V=30.0 PL=1
CALL JOB:EXTRUDE
MOVL C00602 V=30.0 PL=1
CALL JOB:EXTRUDE
MOVL C00603 V=30.0 PL=1
CALL JOB:EXTRUDE
MOVL C00604 V=30.0 PL=1
CALL JOB:EXTRUDE
MOVL C00605 V=30.0 PL=1
CALL JOB:EXTRUDE
MOVL C00606 V=30.0 PL=1
CALL JOB:EXTRUDE
MOVL C00607 V=30.0 PL=1
CALL JOB:EXTRUDE
MOVL C00608 V=30.0 PL=1
CALL JOB:EXTRUDE
MOVL C00609 V=30.0 PL=1
CALL JOB:EXTRUDE
MOVL C00610 V=30.0 PL=1
CALL JOB:EXTRUDE
MOVL C00611 V=30.0 PL=1
CALL JOB:EXTRUDE
MOVL C00612 V=30.0 PL=1
CALL JOB:EXTRUDE
MOVL C00613 V=30.0 PL=1
CALL JOB:EXTRUDE
MOVL C00614 V=30.0 PL=1
CALL JOB:EXTRUDE
MOVL C00615 V=30.0 PL=1
CALL JOB:EXTRUDE
MOVL C00616 V=30.0 PL=1
CALL JOB:EXTRUDE
MOVL C00617 V=30.0 PL=1
CALL JOB:EXTRUDE
MOVL C00618 V=30.0 PL=1
CALL JOB:EXTRUDE
MOVL C00619 V=30.0 PL=1
CALL JOB:EXTRUDE
MOVL C00620 V=30.0 PL=1
CALL JOB:EXTRUDE
MOVL C00621 V=30.0 PL=1
CALL JOB:EXTRUDE
MOVL C00622 V=30.0 PL=1
CALL JOB:EXTRUDE
MOVL C00623 V=30.0 PL=1
CALL JOB:EXTRUDE
MOVL C00624 V=30.0 PL=1
CALL JOB:EXTRUDE
MOVL C00625 V=30.0 PL=1
CALL JOB:EXTRUDE
MOVL C00626 V=30.0 PL=1
CALL JOB:EXTRUDE
MOVL C00627 V=30.0 PL=1
CALL JOB:EXTRUDE
MOVL C00628 V=30.0 PL=1
CALL JOB:EXTRUDE
MOVL C00629 V=30.0 PL=1
CALL JOB:EXTRUDE
MOVL C00630 V=30.0 PL=1
CALL JOB:EXTRUDE
MOVL C00631 V=30.0 PL=1
CALL JOB:EXTRUDE
MOVL C00632 V=30.0 PL=1
CALL JOB:EXTRUDE
MOVL C00633 V=30.0 PL=1
CALL JOB:EXTRUDE
MOVL C00634 V=30.0 PL=1
CALL JOB:EXTRUDE
MOVL C00635 V=30.0 PL=1
CALL JOB:EXTRUDE
MOVL C00636 V=30.0 PL=1
CALL JOB:EXTRUDE
MOVL C00637 V=30.0 PL=1
CALL JOB:EXTRUDE
MOVL C00638 V=30.0 PL=1
CALL JOB:EXTRUDE
MOVL C00639 V=30.0 PL=1
CALL JOB:EXTRUDE
MOVL C00640 V=30.0 PL=1
CALL JOB:EXTRUDE
MOVL C00641 V=30.0 PL=1
CALL JOB:EXTRUDE
MOVL C00642 V=30.0 PL=1
CALL JOB:EXTRUDE
MOVL C00643 V=30.0 PL=1
CALL JOB:EXTRUDE
MOVL C00644 V=30.0 PL=1
CALL JOB:EXTRUDE
MOVL C00645 V=30.0 PL=1
CALL JOB:EXTRUDE
MOVL C00646 V=30.0 PL=1
CALL JOB:EXTRUDE
MOVL C00647 V=30.0 PL=1
CALL JOB:EXTRUDE
MOVL C00648 V=30.0 PL=1
CALL JOB:EXTRUDE
MOVL C00649 V=30.0 PL=1
CALL JOB:EXTRUDE
MOVL C00650 V=30.0 PL=1
CALL JOB:EXTRUDE
MOVL C00651 V=30.0 PL=1
CALL JOB:EXTRUDE
MOVL C00652 V=30.0 PL=1
CALL JOB:EXTRUDE
MOVL C00653 V=30.0 PL=1
CALL JOB:EXTRUDE
MOVL C00654 V=30.0 PL=1
CALL JOB:EXTRUDE
MOVL C00655 V=30.0 PL=1
CALL JOB:EXTRUDE
MOVL C00656 V=30.0 PL=1
CALL JOB:EXTRUDE
MOVL C00657 V=30.0 PL=1
CALL JOB:EXTRUDE
MOVL C00658 V=30.0 PL=1
CALL JOB:EXTRUDE
MOVL C00659 V=30.0 PL=1
CALL JOB:EXTRUDE
MOVL C00660 V=30.0 PL=1
CALL JOB:EXTRUDE
MOVL C00661 V=30.0 PL=1
CALL JOB:EXTRUDE
MOVL C00662 V=30.0 PL=1
CALL JOB:EXTRUDE
MOVL C00663 V=30.0 PL=1
CALL JOB:EXTRUDE
MOVL C00664 V=30.0 PL=1
CALL JOB:EXTRUDE
MOVL C00665 V=30.0 PL=1
CALL JOB:EXTRUDE
MOVL C00666 V=30.0 PL=1
CALL JOB:EXTRUDE
MOVL C00667 V=30.0 PL=1
CALL JOB:EXTRUDE
MOVL C00668 V=30.0 PL=1
CALL JOB:EXTRUDE
MOVL C00669 V=30.0 PL=1
CALL JOB:EXTRUDE
MOVL C00670 V=30.0 PL=1
CALL JOB:EXTRUDE
MOVL C00671 V=30.0 PL=1
CALL JOB:EXTRUDE
MOVL C00672 V=30.0 PL=1
CALL JOB:EXTRUDE
MOVL C00673 V=30.0 PL=1
CALL JOB:EXTRUDE
MOVL C00674 V=30.0 PL=1
CALL JOB:EXTRUDE
MOVL C00675 V=30.0 PL=1
CALL JOB:EXTRUDE
MOVL C00676 V=30.0 PL=1
CALL JOB:EXTRUDE
MOVL C00677 V=30.0 PL=1
CALL JOB:EXTRUDE
MOVL C00678 V=30.0 PL=1
CALL JOB:EXTRUDE
MOVL C00679 V=30.0 PL=1
CALL JOB:EXTRUDE
MOVL C00680 V=30.0 PL=1
CALL JOB:EXTRUDE
MOVL C00681 V=30.0 PL=1
CALL JOB:EXTRUDE
MOVL C00682 V=30.0 PL=1
CALL JOB:EXTRUDE
MOVL C00683 V=30.0 PL=1
CALL JOB:EXTRUDE
MOVL C00684 V=30.0 PL=1
CALL JOB:EXTRUDE
MOVL C00685 V=30.0 PL=1
CALL JOB:EXTRUDE
MOVL C00686 V=30.0 PL=1
CALL JOB:EXTRUDE
MOVL C00687 V=30.0 PL=1
CALL JOB:EXTRUDE
MOVL C00688 V=30.0 PL=1
CALL JOB:EXTRUDE
MOVL C00689 V=30.0 PL=1
CALL JOB:EXTRUDE
MOVL C00690 V=30.0 PL=1
CALL JOB:EXTRUDE
MOVL C00691 V=30.0 PL=1
CALL JOB:EXTRUDE
MOVL C00692 V=30.0 PL=1
MOVL C00693 V=130.0 PL=1
CALL JOB:EXTRUDE
MOVL C00694 V=20.0 PL=1
MOVL C00695 V=130.0 PL=1
CALL JOB:EXTRUDE
MOVL C00696 V=20.0 PL=1
CALL JOB:EXTRUDE
MOVL C00697 V=20.0 PL=1
CALL JOB:EXTRUDE
MOVL C00698 V=20.0 PL=1
CALL JOB:EXTRUDE
MOVL C00699 V=20.0 PL=1
CALL JOB:EXTRUDE
MOVL C00700 V=20.0 PL=1
CALL JOB:EXTRUDE
MOVL C00701 V=20.0 PL=1
CALL JOB:EXTRUDE
MOVL C00702 V=20.0 PL=1
CALL JOB:EXTRUDE
MOVL C00703 V=20.0 PL=1
CALL JOB:EXTRUDE
MOVL C00704 V=20.0 PL=1
CALL JOB:EXTRUDE
MOVL C00705 V=20.0 PL=1
CALL JOB:EXTRUDE
MOVL C00706 V=20.0 PL=1
CALL JOB:EXTRUDE
MOVL C00707 V=20.0 PL=1
CALL JOB:EXTRUDE
MOVL C00708 V=20.0 PL=1
CALL JOB:EXTRUDE
MOVL C00709 V=20.0 PL=1
CALL JOB:EXTRUDE
MOVL C00710 V=20.0 PL=1
CALL JOB:EXTRUDE
MOVL C00711 V=20.0 PL=1
CALL JOB:EXTRUDE
MOVL C00712 V=20.0 PL=1
CALL JOB:EXTRUDE
MOVL C00713 V=20.0 PL=1
CALL JOB:EXTRUDE
MOVL C00714 V=20.0 PL=1
CALL JOB:EXTRUDE
MOVL C00715 V=20.0 PL=1
CALL JOB:EXTRUDE
MOVL C00716 V=20.0 PL=1
CALL JOB:EXTRUDE
MOVL C00717 V=20.0 PL=1
CALL JOB:EXTRUDE
MOVL C00718 V=20.0 PL=1
CALL JOB:EXTRUDE
MOVL C00719 V=20.0 PL=1
CALL JOB:EXTRUDE
MOVL C00720 V=20.0 PL=1
CALL JOB:EXTRUDE
MOVL C00721 V=20.0 PL=1
CALL JOB:EXTRUDE
MOVL C00722 V=20.0 PL=1
CALL JOB:EXTRUDE
MOVL C00723 V=20.0 PL=1
CALL JOB:EXTRUDE
MOVL C00724 V=20.0 PL=1
CALL JOB:EXTRUDE
MOVL C00725 V=20.0 PL=1
CALL JOB:EXTRUDE
MOVL C00726 V=20.0 PL=1
CALL JOB:EXTRUDE
MOVL C00727 V=20.0 PL=1
CALL JOB:EXTRUDE
MOVL C00728 V=20.0 PL=1
CALL JOB:EXTRUDE
MOVL C00729 V=20.0 PL=1
CALL JOB:EXTRUDE
MOVL C00730 V=20.0 PL=1
CALL JOB:EXTRUDE
MOVL C00731 V=20.0 PL=1
CALL JOB:EXTRUDE
MOVL C00732 V=20.0 PL=1
CALL JOB:EXTRUDE
MOVL C00733 V=20.0 PL=1
CALL JOB:EXTRUDE
MOVL C00734 V=20.0 PL=1
CALL JOB:EXTRUDE
MOVL C00735 V=20.0 PL=1
CALL JOB:EXTRUDE
MOVL C00736 V=20.0 PL=1
CALL JOB:EXTRUDE
MOVL C00737 V=20.0 PL=1
CALL JOB:EXTRUDE
MOVL C00738 V=20.0 PL=1
MOVL C00739 V=130.0 PL=1
MOVL C00740 V=130.0 PL=1
CALL JOB:EXTRUDE
MOVL C00741 V=60.0 PL=1
CALL JOB:EXTRUDE
MOVL C00742 V=60.0 PL=1
CALL JOB:EXTRUDE
MOVL C00743 V=60.0 PL=1
CALL JOB:EXTRUDE
MOVL C00744 V=60.0 PL=1
CALL JOB:EXTRUDE
MOVL C00745 V=60.0 PL=1
CALL JOB:EXTRUDE
MOVL C00746 V=60.0 PL=1
CALL JOB:EXTRUDE
MOVL C00747 V=60.0 PL=1
CALL JOB:EXTRUDE
MOVL C00748 V=60.0 PL=1
CALL JOB:EXTRUDE
MOVL C00749 V=60.0 PL=1
CALL JOB:EXTRUDE
MOVL C00750 V=60.0 PL=1
CALL JOB:EXTRUDE
MOVL C00751 V=60.0 PL=1
CALL JOB:EXTRUDE
MOVL C00752 V=60.0 PL=1
CALL JOB:EXTRUDE
MOVL C00753 V=60.0 PL=1
CALL JOB:EXTRUDE
MOVL C00754 V=60.0 PL=1
CALL JOB:EXTRUDE
MOVL C00755 V=60.0 PL=1
CALL JOB:EXTRUDE
MOVL C00756 V=60.0 PL=1
CALL JOB:EXTRUDE
MOVL C00757 V=60.0 PL=1
CALL JOB:EXTRUDE
MOVL C00758 V=60.0 PL=1
CALL JOB:EXTRUDE
MOVL C00759 V=60.0 PL=1
CALL JOB:EXTRUDE
MOVL C00760 V=60.0 PL=1
CALL JOB:EXTRUDE
MOVL C00761 V=60.0 PL=1
CALL JOB:EXTRUDE
MOVL C00762 V=60.0 PL=1
CALL JOB:EXTRUDE
MOVL C00763 V=60.0 PL=1
CALL JOB:EXTRUDE
MOVL C00764 V=60.0 PL=1
MOVL C00765 V=130.0 PL=1
CALL JOB:EXTRUDE
MOVL C00766 V=60.0 PL=1
CALL JOB:EXTRUDE
MOVL C00767 V=60.0 PL=1
CALL JOB:EXTRUDE
MOVL C00768 V=60.0 PL=1
CALL JOB:EXTRUDE
MOVL C00769 V=60.0 PL=1
CALL JOB:EXTRUDE
MOVL C00770 V=60.0 PL=1
CALL JOB:EXTRUDE
MOVL C00771 V=60.0 PL=1
CALL JOB:EXTRUDE
MOVL C00772 V=60.0 PL=1
CALL JOB:EXTRUDE
MOVL C00773 V=60.0 PL=1
CALL JOB:EXTRUDE
MOVL C00774 V=60.0 PL=1
CALL JOB:EXTRUDE
MOVL C00775 V=60.0 PL=1
CALL JOB:EXTRUDE
MOVL C00776 V=60.0 PL=1
CALL JOB:EXTRUDE
MOVL C00777 V=60.0 PL=1
CALL JOB:EXTRUDE
MOVL C00778 V=60.0 PL=1
CALL JOB:EXTRUDE
MOVL C00779 V=60.0 PL=1
CALL JOB:EXTRUDE
MOVL C00780 V=60.0 PL=1
CALL JOB:EXTRUDE
MOVL C00781 V=60.0 PL=1
CALL JOB:EXTRUDE
MOVL C00782 V=60.0 PL=1
CALL JOB:EXTRUDE
MOVL C00783 V=60.0 PL=1
CALL JOB:EXTRUDE
MOVL C00784 V=60.0 PL=1
CALL JOB:EXTRUDE
MOVL C00785 V=60.0 PL=1
CALL JOB:EXTRUDE
MOVL C00786 V=60.0 PL=1
CALL JOB:EXTRUDE
MOVL C00787 V=60.0 PL=1
CALL JOB:EXTRUDE
MOVL C00788 V=60.0 PL=1
CALL JOB:EXTRUDE
MOVL C00789 V=60.0 PL=1
CALL JOB:EXTRUDE
MOVL C00790 V=60.0 PL=1
CALL JOB:EXTRUDE
MOVL C00791 V=60.0 PL=1
CALL JOB:EXTRUDE
MOVL C00792 V=60.0 PL=1
CALL JOB:EXTRUDE
MOVL C00793 V=60.0 PL=1
CALL JOB:EXTRUDE
MOVL C00794 V=60.0 PL=1
CALL JOB:EXTRUDE
MOVL C00795 V=60.0 PL=1
CALL JOB:EXTRUDE
MOVL C00796 V=60.0 PL=1
CALL JOB:EXTRUDE
MOVL C00797 V=60.0 PL=1
CALL JOB:EXTRUDE
MOVL C00798 V=60.0 PL=1
CALL JOB:EXTRUDE
MOVL C00799 V=60.0 PL=1
CALL JOB:EXTRUDE
MOVL C00800 V=60.0 PL=1
CALL JOB:EXTRUDE
MOVL C00801 V=60.0 PL=1
CALL JOB:EXTRUDE
MOVL C00802 V=60.0 PL=1
CALL JOB:EXTRUDE
MOVL C00803 V=60.0 PL=1
CALL JOB:EXTRUDE
MOVL C00804 V=60.0 PL=1
CALL JOB:EXTRUDE
MOVL C00805 V=60.0 PL=1
CALL JOB:EXTRUDE
MOVL C00806 V=60.0 PL=1
CALL JOB:EXTRUDE
MOVL C00807 V=60.0 PL=1
MOVL C00808 V=130.0 PL=1
CALL JOB:EXTRUDE
MOVL C00809 V=30.0 PL=1
CALL JOB:EXTRUDE
MOVL C00810 V=30.0 PL=1
CALL JOB:EXTRUDE
MOVL C00811 V=30.0 PL=1
CALL JOB:EXTRUDE
MOVL C00812 V=30.0 PL=1
CALL JOB:EXTRUDE
MOVL C00813 V=30.0 PL=1
CALL JOB:EXTRUDE
MOVL C00814 V=30.0 PL=1
CALL JOB:EXTRUDE
MOVL C00815 V=30.0 PL=1
CALL JOB:EXTRUDE
MOVL C00816 V=30.0 PL=1
CALL JOB:EXTRUDE
MOVL C00817 V=30.0 PL=1
CALL JOB:EXTRUDE
MOVL C00818 V=30.0 PL=1
CALL JOB:EXTRUDE
MOVL C00819 V=30.0 PL=1
CALL JOB:EXTRUDE
MOVL C00820 V=30.0 PL=1
CALL JOB:EXTRUDE
MOVL C00821 V=30.0 PL=1
CALL JOB:EXTRUDE
MOVL C00822 V=30.0 PL=1
CALL JOB:EXTRUDE
MOVL C00823 V=30.0 PL=1
CALL JOB:EXTRUDE
MOVL C00824 V=30.0 PL=1
CALL JOB:EXTRUDE
MOVL C00825 V=30.0 PL=1
CALL JOB:EXTRUDE
MOVL C00826 V=30.0 PL=1
CALL JOB:EXTRUDE
MOVL C00827 V=30.0 PL=1
CALL JOB:EXTRUDE
MOVL C00828 V=30.0 PL=1
CALL JOB:EXTRUDE
MOVL C00829 V=30.0 PL=1
CALL JOB:EXTRUDE
MOVL C00830 V=30.0 PL=1
CALL JOB:EXTRUDE
MOVL C00831 V=30.0 PL=1
CALL JOB:EXTRUDE
MOVL C00832 V=30.0 PL=1
CALL JOB:EXTRUDE
MOVL C00833 V=30.0 PL=1
CALL JOB:EXTRUDE
MOVL C00834 V=30.0 PL=1
CALL JOB:EXTRUDE
MOVL C00835 V=30.0 PL=1
CALL JOB:EXTRUDE
MOVL C00836 V=30.0 PL=1
CALL JOB:EXTRUDE
MOVL C00837 V=30.0 PL=1
CALL JOB:EXTRUDE
MOVL C00838 V=30.0 PL=1
CALL JOB:EXTRUDE
MOVL C00839 V=30.0 PL=1
CALL JOB:EXTRUDE
MOVL C00840 V=30.0 PL=1
CALL JOB:EXTRUDE
MOVL C00841 V=30.0 PL=1
CALL JOB:EXTRUDE
MOVL C00842 V=30.0 PL=1
CALL JOB:EXTRUDE
MOVL C00843 V=30.0 PL=1
CALL JOB:EXTRUDE
MOVL C00844 V=30.0 PL=1
CALL JOB:EXTRUDE
MOVL C00845 V=30.0 PL=1
CALL JOB:EXTRUDE
MOVL C00846 V=30.0 PL=1
CALL JOB:EXTRUDE
MOVL C00847 V=30.0 PL=1
CALL JOB:EXTRUDE
MOVL C00848 V=30.0 PL=1
CALL JOB:EXTRUDE
MOVL C00849 V=30.0 PL=1
CALL JOB:EXTRUDE
MOVL C00850 V=30.0 PL=1
CALL JOB:EXTRUDE
MOVL C00851 V=30.0 PL=1
CALL JOB:EXTRUDE
MOVL C00852 V=30.0 PL=1
CALL JOB:EXTRUDE
MOVL C00853 V=30.0 PL=1
CALL JOB:EXTRUDE
MOVL C00854 V=30.0 PL=1
CALL JOB:EXTRUDE
MOVL C00855 V=30.0 PL=1
CALL JOB:EXTRUDE
MOVL C00856 V=30.0 PL=1
CALL JOB:EXTRUDE
MOVL C00857 V=30.0 PL=1
CALL JOB:EXTRUDE
MOVL C00858 V=30.0 PL=1
CALL JOB:EXTRUDE
MOVL C00859 V=30.0 PL=1
CALL JOB:EXTRUDE
MOVL C00860 V=30.0 PL=1
CALL JOB:EXTRUDE
MOVL C00861 V=30.0 PL=1
CALL JOB:EXTRUDE
MOVL C00862 V=30.0 PL=1
CALL JOB:EXTRUDE
MOVL C00863 V=30.0 PL=1
CALL JOB:EXTRUDE
MOVL C00864 V=30.0 PL=1
CALL JOB:EXTRUDE
MOVL C00865 V=30.0 PL=1
CALL JOB:EXTRUDE
MOVL C00866 V=30.0 PL=1
CALL JOB:EXTRUDE
MOVL C00867 V=30.0 PL=1
CALL JOB:EXTRUDE
MOVL C00868 V=30.0 PL=1
CALL JOB:EXTRUDE
MOVL C00869 V=30.0 PL=1
CALL JOB:EXTRUDE
MOVL C00870 V=30.0 PL=1
CALL JOB:EXTRUDE
MOVL C00871 V=30.0 PL=1
CALL JOB:EXTRUDE
MOVL C00872 V=30.0 PL=1
CALL JOB:EXTRUDE
MOVL C00873 V=30.0 PL=1
CALL JOB:EXTRUDE
MOVL C00874 V=30.0 PL=1
CALL JOB:EXTRUDE
MOVL C00875 V=30.0 PL=1
CALL JOB:EXTRUDE
MOVL C00876 V=30.0 PL=1
CALL JOB:EXTRUDE
MOVL C00877 V=30.0 PL=1
CALL JOB:EXTRUDE
MOVL C00878 V=30.0 PL=1
CALL JOB:EXTRUDE
MOVL C00879 V=30.0 PL=1
CALL JOB:EXTRUDE
MOVL C00880 V=30.0 PL=1
MOVL C00881 V=130.0 PL=1
CALL JOB:EXTRUDE
CALL JOB:EXTRUDE
MOVL C00882 V=130.0 PL=1
CALL JOB:EXTRUDE
CALL JOB:EXTRUDE
MOVL C00883 V=30.0 PL=1
CALL JOB:EXTRUDE
MOVL C00884 V=30.0 PL=1
CALL JOB:EXTRUDE
MOVL C00885 V=30.0 PL=1
CALL JOB:EXTRUDE
MOVL C00886 V=30.0 PL=1
CALL JOB:EXTRUDE
MOVL C00887 V=30.0 PL=1
CALL JOB:EXTRUDE
MOVL C00888 V=30.0 PL=1
CALL JOB:EXTRUDE
MOVL C00889 V=30.0 PL=1
CALL JOB:EXTRUDE
MOVL C00890 V=30.0 PL=1
CALL JOB:EXTRUDE
MOVL C00891 V=30.0 PL=1
CALL JOB:EXTRUDE
MOVL C00892 V=30.0 PL=1
CALL JOB:EXTRUDE
MOVL C00893 V=30.0 PL=1
CALL JOB:EXTRUDE
MOVL C00894 V=30.0 PL=1
CALL JOB:EXTRUDE
MOVL C00895 V=30.0 PL=1
CALL JOB:EXTRUDE
MOVL C00896 V=30.0 PL=1
CALL JOB:EXTRUDE
MOVL C00897 V=30.0 PL=1
CALL JOB:EXTRUDE
MOVL C00898 V=30.0 PL=1
CALL JOB:EXTRUDE
MOVL C00899 V=30.0 PL=1
CALL JOB:EXTRUDE
MOVL C00900 V=30.0 PL=1
CALL JOB:EXTRUDE
MOVL C00901 V=30.0 PL=1
CALL JOB:EXTRUDE
MOVL C00902 V=30.0 PL=1
CALL JOB:EXTRUDE
MOVL C00903 V=30.0 PL=1
CALL JOB:EXTRUDE
MOVL C00904 V=30.0 PL=1
CALL JOB:EXTRUDE
MOVL C00905 V=30.0 PL=1
CALL JOB:EXTRUDE
MOVL C00906 V=30.0 PL=1
CALL JOB:EXTRUDE
MOVL C00907 V=30.0 PL=1
CALL JOB:EXTRUDE
MOVL C00908 V=30.0 PL=1
CALL JOB:EXTRUDE
MOVL C00909 V=30.0 PL=1
CALL JOB:EXTRUDE
MOVL C00910 V=30.0 PL=1
CALL JOB:EXTRUDE
MOVL C00911 V=30.0 PL=1
CALL JOB:EXTRUDE
MOVL C00912 V=30.0 PL=1
CALL JOB:EXTRUDE
MOVL C00913 V=30.0 PL=1
CALL JOB:EXTRUDE
MOVL C00914 V=30.0 PL=1
CALL JOB:EXTRUDE
MOVL C00915 V=30.0 PL=1
CALL JOB:EXTRUDE
MOVL C00916 V=30.0 PL=1
CALL JOB:EXTRUDE
MOVL C00917 V=30.0 PL=1
CALL JOB:EXTRUDE
MOVL C00918 V=30.0 PL=1
CALL JOB:EXTRUDE
MOVL C00919 V=30.0 PL=1
CALL JOB:EXTRUDE
MOVL C00920 V=30.0 PL=1
CALL JOB:EXTRUDE
MOVL C00921 V=30.0 PL=1
CALL JOB:EXTRUDE
MOVL C00922 V=30.0 PL=1
CALL JOB:EXTRUDE
MOVL C00923 V=30.0 PL=1
CALL JOB:EXTRUDE
MOVL C00924 V=30.0 PL=1
CALL JOB:EXTRUDE
MOVL C00925 V=30.0 PL=1
CALL JOB:EXTRUDE
MOVL C00926 V=30.0 PL=1
CALL JOB:EXTRUDE
MOVL C00927 V=30.0 PL=1
CALL JOB:EXTRUDE
MOVL C00928 V=30.0 PL=1
CALL JOB:EXTRUDE
MOVL C00929 V=30.0 PL=1
CALL JOB:EXTRUDE
MOVL C00930 V=30.0 PL=1
CALL JOB:EXTRUDE
MOVL C00931 V=30.0 PL=1
CALL JOB:EXTRUDE
MOVL C00932 V=30.0 PL=1
CALL JOB:EXTRUDE
MOVL C00933 V=30.0 PL=1
CALL JOB:EXTRUDE
MOVL C00934 V=30.0 PL=1
CALL JOB:EXTRUDE
MOVL C00935 V=30.0 PL=1
CALL JOB:EXTRUDE
MOVL C00936 V=30.0 PL=1
CALL JOB:EXTRUDE
MOVL C00937 V=30.0 PL=1
CALL JOB:EXTRUDE
MOVL C00938 V=30.0 PL=1
CALL JOB:EXTRUDE
MOVL C00939 V=30.0 PL=1
CALL JOB:EXTRUDE
MOVL C00940 V=30.0 PL=1
CALL JOB:EXTRUDE
MOVL C00941 V=30.0 PL=1
CALL JOB:EXTRUDE
MOVL C00942 V=30.0 PL=1
CALL JOB:EXTRUDE
MOVL C00943 V=30.0 PL=1
CALL JOB:EXTRUDE
MOVL C00944 V=30.0 PL=1
CALL JOB:EXTRUDE
MOVL C00945 V=30.0 PL=1
CALL JOB:EXTRUDE
MOVL C00946 V=30.0 PL=1
CALL JOB:EXTRUDE
MOVL C00947 V=30.0 PL=1
CALL JOB:EXTRUDE
MOVL C00948 V=30.0 PL=1
CALL JOB:EXTRUDE
MOVL C00949 V=30.0 PL=1
CALL JOB:EXTRUDE
MOVL C00950 V=30.0 PL=1
CALL JOB:EXTRUDE
MOVL C00951 V=30.0 PL=1
CALL JOB:EXTRUDE
MOVL C00952 V=30.0 PL=1
CALL JOB:EXTRUDE
MOVL C00953 V=30.0 PL=1
CALL JOB:EXTRUDE
MOVL C00954 V=30.0 PL=1
CALL JOB:EXTRUDE
MOVL C00955 V=30.0 PL=1
CALL JOB:EXTRUDE
MOVL C00956 V=30.0 PL=1
CALL JOB:EXTRUDE
MOVL C00957 V=30.0 PL=1
CALL JOB:EXTRUDE
MOVL C00958 V=30.0 PL=1
CALL JOB:EXTRUDE
MOVL C00959 V=30.0 PL=1
CALL JOB:EXTRUDE
MOVL C00960 V=30.0 PL=1
CALL JOB:EXTRUDE
MOVL C00961 V=30.0 PL=1
CALL JOB:EXTRUDE
MOVL C00962 V=30.0 PL=1
CALL JOB:EXTRUDE
MOVL C00963 V=30.0 PL=1
CALL JOB:EXTRUDE
MOVL C00964 V=30.0 PL=1
CALL JOB:EXTRUDE
MOVL C00965 V=30.0 PL=1
CALL JOB:EXTRUDE
MOVL C00966 V=30.0 PL=1
CALL JOB:EXTRUDE
MOVL C00967 V=30.0 PL=1
CALL JOB:EXTRUDE
MOVL C00968 V=30.0 PL=1
CALL JOB:EXTRUDE
MOVL C00969 V=30.0 PL=1
CALL JOB:EXTRUDE
MOVL C00970 V=30.0 PL=1
CALL JOB:EXTRUDE
MOVL C00971 V=30.0 PL=1
CALL JOB:EXTRUDE
MOVL C00972 V=30.0 PL=1
CALL JOB:EXTRUDE
MOVL C00973 V=30.0 PL=1
CALL JOB:EXTRUDE
MOVL C00974 V=30.0 PL=1
CALL JOB:EXTRUDE
MOVL C00975 V=30.0 PL=1
CALL JOB:EXTRUDE
MOVL C00976 V=30.0 PL=1
CALL JOB:EXTRUDE
MOVL C00977 V=30.0 PL=1
CALL JOB:EXTRUDE
MOVL C00978 V=30.0 PL=1
CALL JOB:EXTRUDE
MOVL C00979 V=30.0 PL=1
CALL JOB:EXTRUDE
MOVL C00980 V=30.0 PL=1
CALL JOB:EXTRUDE
MOVL C00981 V=30.0 PL=1
CALL JOB:EXTRUDE
MOVL C00982 V=30.0 PL=1
CALL JOB:EXTRUDE
MOVL C00983 V=30.0 PL=1
CALL JOB:EXTRUDE
MOVL C00984 V=30.0 PL=1
CALL JOB:EXTRUDE
MOVL C00985 V=30.0 PL=1
CALL JOB:EXTRUDE
MOVL C00986 V=30.0 PL=1
CALL JOB:EXTRUDE
MOVL C00987 V=30.0 PL=1
CALL JOB:EXTRUDE
MOVL C00988 V=30.0 PL=1
CALL JOB:EXTRUDE
MOVL C00989 V=30.0 PL=1
CALL JOB:EXTRUDE
MOVL C00990 V=30.0 PL=1
CALL JOB:EXTRUDE
MOVL C00991 V=30.0 PL=1
CALL JOB:EXTRUDE
MOVL C00992 V=30.0 PL=1
CALL JOB:EXTRUDE
MOVL C00993 V=30.0 PL=1
CALL JOB:EXTRUDE
CALL JOB:EXTRUDE
MOVL C00994 V=130.0 PL=1
CALL JOB:EXTRUDE
CALL JOB:EXTRUDE
MOVL C00995 V=30.0 PL=1
CALL JOB:EXTRUDE
MOVL C00996 V=30.0 PL=1
CALL JOB:EXTRUDE
MOVL C00997 V=30.0 PL=1
CALL JOB:EXTRUDE
MOVL C00998 V=30.0 PL=1
CALL JOB:EXTRUDE
END
